LIN {X 0,Y 364.847,Z 1093.089,A -85,B 0,C 180,E1 16368.459,E2 16368.459} C_VEL
LIN {X 0,Y 364.189,Z 1097.02,A -85,B 0,C 180,E1 16366.666,E2 16366.666} C_VEL
LIN {X 0,Y 363.606,Z 1099.933,A -85,B 0,C 180,E1 16364.529,E2 16364.529} C_VEL
LIN {X 0,Y 363.242,Z 1100.889,A -85,B 0,C 180,E1 16362.54,E2 16362.54} C_VEL
LIN {X 0,Y 363.064,Z 1100.469,A -85,B 0,C 180,E1 16360.702,E2 16360.702} C_VEL
LIN {X 0,Y 363.041,Z 1098.768,A -85,B 0,C 180,E1 16358.85,E2 16358.85} C_VEL
LIN {X 0,Y 363.189,Z 1095.43,A -85,B 0,C 180,E1 16356.816,E2 16356.816} C_VEL
LIN {X 0,Y 363.562,Z 1089.731,A -85,B 0,C 180,E1 16354.593,E2 16354.593} C_VEL
LIN {X 0,Y 364.021,Z 1083.743,A -85,B 0,C 180,E1 16352.871,E2 16352.871} C_VEL
LIN {X 0,Y 364.565,Z 1076.974,A -85,B 0,C 180,E1 16351.316,E2 16351.316} C_VEL
LIN {X 0,Y 365.337,Z 1067.492,A -85,B 0,C 180,E1 16349.558,E2 16349.558} C_VEL
LIN {X 0,Y 366.143,Z 1056.281,A -85,B 0,C 180,E1 16347.95,E2 16347.95} C_VEL
LIN {X 0,Y 366.856,Z 1045.383,A -85,B 0,C 180,E1 16346.688,E2 16346.688} C_VEL
LIN {X 0,Y 366.982,Z 1044.003,A -85,B 0,C 180,E1 16346.513,E2 16346.513} C_VEL
LIN {X 0,Y 368.446,Z 1044.428,A -85,B 0,C 180,E1 16346.01,E2 16346.01} C_VEL
LIN {X 0,Y 371.071,Z 1043.748,A -85,B 0,C 180,E1 16345.537,E2 16345.537} C_VEL
LIN {X 0,Y 374.017,Z 1043.467,A -85,B 0,C 180,E1 16344.893,E2 16344.893} C_VEL
LIN {X 0,Y 377.167,Z 1042.77,A -85,B 0,C 180,E1 16344.322,E2 16344.322} C_VEL
LIN {X 0,Y 386.849,Z 1040.234,A -85,B 0,C 180,E1 16342.784,E2 16342.784} C_VEL
LIN {X 0,Y 400.514,Z 1035.789,A -85,B 0,C 180,E1 16341.014,E2 16341.014} C_VEL
LIN {X 0,Y 412.392,Z 1030.85,A -85,B 0,C 180,E1 16339.838,E2 16339.838} C_VEL
LIN {X 0,Y 415.714,Z 1029.331,A -85,B 0,C 180,E1 16339.543,E2 16339.543} C_VEL
LIN {X 0,Y 407.381,Z 1049.235,A -85,B 0,C 180,E1 16337.007,E2 16337.007} C_VEL
LIN {X 0,Y 399.448,Z 1067.755,A -85,B 0,C 180,E1 16334.282,E2 16334.282} C_VEL
LIN {X 0,Y 391.606,Z 1085.492,A -85,B 0,C 180,E1 16331.206,E2 16331.206} C_VEL
LIN {X 0,Y 384.418,Z 1102.08,A -85,B 0,C 180,E1 16327.87,E2 16327.87} C_VEL
LIN {X 0,Y 378.236,Z 1116.473,A -85,B 0,C 180,E1 16324.454,E2 16324.454} C_VEL
LIN {X 0,Y 372.918,Z 1129.743,A -85,B 0,C 180,E1 16320.807,E2 16320.807} C_VEL
LIN {X 0,Y 368.629,Z 1141.026,A -85,B 0,C 180,E1 16317.111,E2 16317.111} C_VEL
LIN {X 0,Y 365.504,Z 1150.37,A -85,B 0,C 180,E1 16313.543,E2 16313.543} C_VEL
LIN {X 0,Y 362.854,Z 1159.499,A -85,B 0,C 180,E1 16309.311,E2 16309.311} C_VEL
LIN {X 0,Y 361.475,Z 1165.476,A -85,B 0,C 180,E1 16305.895,E2 16305.895} C_VEL
LIN {X 0,Y 360.647,Z 1170.154,A -85,B 0,C 180,E1 16302.599,E2 16302.599} C_VEL
LIN {X 0,Y 360.167,Z 1174.441,A -85,B 0,C 180,E1 16298.624,E2 16298.624} C_VEL
LIN {X 0,Y 359.992,Z 1176.868,A -85,B 0,C 180,E1 16294.941,E2 16294.941} C_VEL
LIN {X 0,Y 359.958,Z 1177.939,A -85,B 0,C 180,E1 16291.753,E2 16291.753} C_VEL
LIN {X 0,Y 359.957,Z 1178.023,A -85,B 0,C 180,E1 16288.729,E2 16288.729} C_VEL
LIN {X 0,Y 359.981,Z 1177.183,A -85,B 0,C 180,E1 16285.689,E2 16285.689} C_VEL
LIN {X 0,Y 360.071,Z 1175.437,A -85,B 0,C 180,E1 16282.663,E2 16282.663} C_VEL
LIN {X 0,Y 360.313,Z 1172.766,A -85,B 0,C 180,E1 16279.61,E2 16279.61} C_VEL
LIN {X 0,Y 360.88,Z 1168.742,A -85,B 0,C 180,E1 16276.217,E2 16276.217} C_VEL
LIN {X 0,Y 361.623,Z 1164.805,A -85,B 0,C 180,E1 16273.586,E2 16273.586} C_VEL
LIN {X 0,Y 361.083,Z 1162.995,A -85,B 0,C 180,E1 16272.394,E2 16272.394} C_VEL
LIN {X 0,Y 356.335,Z 1157.659,A -85,B 0,C 180,E1 16269.097,E2 16269.097} C_VEL
LIN {X 0,Y 356.258,Z 1155.765,A -85,B 0,C 180,E1 16268.158,E2 16268.158} C_VEL
LIN {X 0,Y 358.806,Z 1148.037,A -85,B 0,C 180,E1 16264.765,E2 16264.765} C_VEL
LIN {X 0,Y 362.973,Z 1136.898,A -85,B 0,C 180,E1 16260.64,E2 16260.64} C_VEL
LIN {X 0,Y 367.709,Z 1125.312,A -85,B 0,C 180,E1 16257.057,E2 16257.057} C_VEL
LIN {X 0,Y 373.773,Z 1111.505,A -85,B 0,C 180,E1 16253.374,E2 16253.374} C_VEL
LIN {X 0,Y 380.314,Z 1096.941,A -85,B 0,C 180,E1 16250.099,E2 16250.099} C_VEL
LIN {X 0,Y 387.848,Z 1080.633,A -85,B 0,C 180,E1 16246.911,E2 16246.911} C_VEL
LIN {X 0,Y 395.874,Z 1062.8,A -85,B 0,C 180,E1 16243.962,E2 16243.962} C_VEL
LIN {X 0,Y 403.958,Z 1044.778,A -85,B 0,C 180,E1 16241.368,E2 16241.368} C_VEL
LIN {X 0,Y 412.483,Z 1024.657,A -85,B 0,C 180,E1 16238.914,E2 16238.914} C_VEL
LIN {X 0,Y 421.011,Z 1003.86,A -85,B 0,C 180,E1 16236.726,E2 16236.726} C_VEL
LIN {X 0,Y 429.064,Z 982.412,A -85,B 0,C 180,E1 16234.817,E2 16234.817} C_VEL
LIN {X 0,Y 436.879,Z 960.16,A -85,B 0,C 180,E1 16233.11,E2 16233.11} C_VEL
LIN {X 0,Y 443.975,Z 937.444,A -85,B 0,C 180,E1 16231.651,E2 16231.651} C_VEL
LIN {X 0,Y 450.439,Z 914.796,A -85,B 0,C 180,E1 16230.406,E2 16230.406} C_VEL
LIN {X 0,Y 456.319,Z 890.425,A -85,B 0,C 180,E1 16229.301,E2 16229.301} C_VEL
LIN {X 0,Y 461.547,Z 865.497,A -85,B 0,C 180,E1 16228.371,E2 16228.371} C_VEL
LIN {X 0,Y 467.573,Z 829.912,A -85,B 0,C 180,E1 16227.349,E2 16227.349} C_VEL
LIN {X 0,Y 480.681,Z 750.241,A -85,B 0,C 180,E1 16225.486,E2 16225.486} C_VEL
LIN {X 0,Y 491.44,Z 677.516,A -85,B 0,C 180,E1 16223.979,E2 16223.979} C_VEL
LIN {X 0,Y 500.182,Z 608.907,A -85,B 0,C 180,E1 16222.702,E2 16222.702} C_VEL
LIN {X 0,Y 506.001,Z 552.806,A -85,B 0,C 180,E1 16221.724,E2 16221.724} C_VEL
LIN {X 0,Y 502.096,Z 549.766,A -85,B 0,C 180,E1 16220.396,E2 16220.396} C_VEL
LIN {X 0,Y 494.551,Z 544.225,A -85,B 0,C 180,E1 16217.533,E2 16217.533} C_VEL
LIN {X 0,Y 486.719,Z 540.701,A -85,B 0,C 180,E1 16214.029,E2 16214.029} C_VEL
LIN {X 0,Y 480.667,Z 539.029,A -85,B 0,C 180,E1 16210.548,E2 16210.548} C_VEL
LIN {X 0,Y 479.161,Z 538.841,A -85,B 0,C 180,E1 16209.489,E2 16209.489} C_VEL
LIN {X 0,Y 474.514,Z 541.062,A -85,B 0,C 180,E1 16205.32,E2 16205.32} C_VEL
LIN {X 0,Y 472.587,Z 544.325,A -85,B 0,C 180,E1 16202.425,E2 16202.425} C_VEL
LIN {X 0,Y 471.775,Z 549.574,A -85,B 0,C 180,E1 16199.15,E2 16199.15} C_VEL
LIN {X 0,Y 474.61,Z 557.775,A -85,B 0,C 180,E1 16195.892,E2 16195.892} C_VEL
LIN {X 0,Y 476.871,Z 565.149,A -85,B 0,C 180,E1 16193.499,E2 16193.499} C_VEL
LIN {X 0,Y 472.618,Z 578.224,A -85,B 0,C 180,E1 16192.256,E2 16192.256} C_VEL
LIN {X 0,Y 471.814,Z 611.299,A -85,B 0,C 180,E1 16189.784,E2 16189.784} C_VEL
LIN {X 0,Y 471.576,Z 643.072,A -85,B 0,C 180,E1 16187.572,E2 16187.572} C_VEL
LIN {X 0,Y 471.999,Z 675.982,A -85,B 0,C 180,E1 16185.281,E2 16185.281} C_VEL
LIN {X 0,Y 473.232,Z 701.845,A -85,B 0,C 180,E1 16183.221,E2 16183.221} C_VEL
LIN {X 0,Y 475.279,Z 724.423,A -85,B 0,C 180,E1 16181.175,E2 16181.175} C_VEL
LIN {X 0,Y 477.851,Z 742.846,A -85,B 0,C 180,E1 16179.323,E2 16179.323} C_VEL
LIN {X 0,Y 481.269,Z 760.271,A -85,B 0,C 180,E1 16177.412,E2 16177.412} C_VEL
LIN {X 0,Y 486.893,Z 780.718,A -85,B 0,C 180,E1 16174.94,E2 16174.94} C_VEL
LIN {X 0,Y 486.96,Z 781.774,A -85,B 0,C 180,E1 16174.871,E2 16174.871} C_VEL
LIN {X 0,Y 480.312,Z 821.81,A -85,B 0,C 180,E1 16174.02,E2 16174.02} C_VEL
LIN {X 0,Y 472.503,Z 860.702,A -85,B 0,C 180,E1 16173.049,E2 16173.049} C_VEL
LIN {X 0,Y 464.769,Z 894.968,A -85,B 0,C 180,E1 16171.953,E2 16171.953} C_VEL
LIN {X 0,Y 456.674,Z 928.359,A -85,B 0,C 180,E1 16170.62,E2 16170.62} C_VEL
LIN {X 0,Y 448.577,Z 959.455,A -85,B 0,C 180,E1 16169.108,E2 16169.108} C_VEL
LIN {X 0,Y 440.535,Z 988.437,A -85,B 0,C 180,E1 16167.433,E2 16167.433} C_VEL
LIN {X 0,Y 433.872,Z 1010.028,A -85,B 0,C 180,E1 16165.943,E2 16165.943} C_VEL
LIN {X 0,Y 426.483,Z 1031.191,A -85,B 0,C 180,E1 16164.209,E2 16164.209} C_VEL
LIN {X 0,Y 419.044,Z 1050.358,A -85,B 0,C 180,E1 16162.349,E2 16162.349} C_VEL
LIN {X 0,Y 411.17,Z 1069.3,A -85,B 0,C 180,E1 16160.211,E2 16160.211} C_VEL
LIN {X 0,Y 402.736,Z 1088.062,A -85,B 0,C 180,E1 16157.716,E2 16157.716} C_VEL
LIN {X 0,Y 394.452,Z 1105.313,A -85,B 0,C 180,E1 16154.989,E2 16154.989} C_VEL
LIN {X 0,Y 386.613,Z 1120.941,A -85,B 0,C 180,E1 16152.075,E2 16152.075} C_VEL
LIN {X 0,Y 378.836,Z 1136.107,A -85,B 0,C 180,E1 16148.718,E2 16148.718} C_VEL
LIN {X 0,Y 371.928,Z 1149.46,A -85,B 0,C 180,E1 16145.187,E2 16145.187} C_VEL
LIN {X 0,Y 365.978,Z 1161.24,A -85,B 0,C 180,E1 16141.452,E2 16141.452} C_VEL
LIN {X 0,Y 360.912,Z 1171.835,A -85,B 0,C 180,E1 16137.378,E2 16137.378} C_VEL
LIN {X 0,Y 357.016,Z 1180.868,A -85,B 0,C 180,E1 16133.082,E2 16133.082} C_VEL
LIN {X 0,Y 354.391,Z 1188.078,A -85,B 0,C 180,E1 16128.76,E2 16128.76} C_VEL
LIN {X 0,Y 352.869,Z 1193.636,A -85,B 0,C 180,E1 16124.437,E2 16124.437} C_VEL
LIN {X 0,Y 352.161,Z 1197.659,A -85,B 0,C 180,E1 16120.137,E2 16120.137} C_VEL
LIN {X 0,Y 351.969,Z 1200.163,A -85,B 0,C 180,E1 16116.031,E2 16116.031} C_VEL
LIN {X 0,Y 351.957,Z 1201.387,A -85,B 0,C 180,E1 16112.115,E2 16112.115} C_VEL
LIN {X 0,Y 351.961,Z 1201.43,A -85,B 0,C 180,E1 16108.37,E2 16108.37} C_VEL
LIN {X 0,Y 351.963,Z 1200.374,A -85,B 0,C 180,E1 16104.455,E2 16104.455} C_VEL
LIN {X 0,Y 352.107,Z 1198.172,A -85,B 0,C 180,E1 16100.518,E2 16100.518} C_VEL
LIN {X 0,Y 352.708,Z 1194.383,A -85,B 0,C 180,E1 16096.222,E2 16096.222} C_VEL
LIN {X 0,Y 354.091,Z 1189.033,A -85,B 0,C 180,E1 16091.902,E2 16091.902} C_VEL
LIN {X 0,Y 356.533,Z 1182.047,A -85,B 0,C 180,E1 16087.577,E2 16087.577} C_VEL
LIN {X 0,Y 360.222,Z 1173.286,A -85,B 0,C 180,E1 16083.276,E2 16083.276} C_VEL
LIN {X 0,Y 365.081,Z 1163.008,A -85,B 0,C 180,E1 16079.191,E2 16079.191} C_VEL
LIN {X 0,Y 371.267,Z 1150.699,A -85,B 0,C 180,E1 16075.181,E2 16075.181} C_VEL
LIN {X 0,Y 378.516,Z 1136.712,A -85,B 0,C 180,E1 16071.432,E2 16071.432} C_VEL
LIN {X 0,Y 386.202,Z 1121.734,A -85,B 0,C 180,E1 16068.088,E2 16068.088} C_VEL
LIN {X 0,Y 394.075,Z 1106.054,A -85,B 0,C 180,E1 16065.139,E2 16065.139} C_VEL
LIN {X 0,Y 402.703,Z 1088.053,A -85,B 0,C 180,E1 16062.29,E2 16062.29} C_VEL
LIN {X 0,Y 410.926,Z 1069.744,A -85,B 0,C 180,E1 16059.851,E2 16059.851} C_VEL
LIN {X 0,Y 419.14,Z 1050.106,A -85,B 0,C 180,E1 16057.625,E2 16057.625} C_VEL
LIN {X 0,Y 427.021,Z 1029.58,A -85,B 0,C 180,E1 16055.656,E2 16055.656} C_VEL
LIN {X 0,Y 434.714,Z 1007.363,A -85,B 0,C 180,E1 16053.865,E2 16053.865} C_VEL
LIN {X 0,Y 441.705,Z 984.375,A -85,B 0,C 180,E1 16052.316,E2 16052.316} C_VEL
LIN {X 0,Y 450.4,Z 952.387,A -85,B 0,C 180,E1 16050.529,E2 16050.529} C_VEL
LIN {X 0,Y 458.422,Z 921.073,A -85,B 0,C 180,E1 16049.07,E2 16049.07} C_VEL
LIN {X 0,Y 466.669,Z 886.521,A -85,B 0,C 180,E1 16047.759,E2 16047.759} C_VEL
LIN {X 0,Y 474.383,Z 851.48,A -85,B 0,C 180,E1 16046.708,E2 16046.708} C_VEL
LIN {X 0,Y 482.278,Z 810.288,A -85,B 0,C 180,E1 16045.722,E2 16045.722} C_VEL
LIN {X 0,Y 488.506,Z 769.42,A -85,B 0,C 180,E1 16044.887,E2 16044.887} C_VEL
LIN {X 0,Y 493.484,Z 727.631,A -85,B 0,C 180,E1 16044.188,E2 16044.188} C_VEL
LIN {X 0,Y 498.328,Z 671.925,A -85,B 0,C 180,E1 16043.44,E2 16043.44} C_VEL
LIN {X 0,Y 501.803,Z 632.657,A -85,B 0,C 180,E1 16042.905,E2 16042.905} C_VEL
LIN {X 0,Y 505.015,Z 611.369,A -85,B 0,C 180,E1 16042.605,E2 16042.605} C_VEL
LIN {X 0,Y 498.401,Z 626.921,A -85,B 0,C 180,E1 16041.748,E2 16041.748} C_VEL
LIN {X 0,Y 492.948,Z 644.379,A -85,B 0,C 180,E1 16040.916,E2 16040.916} C_VEL
LIN {X 0,Y 489.241,Z 656.284,A -85,B 0,C 180,E1 16040.254,E2 16040.254} C_VEL
LIN {X 0,Y 483.115,Z 679.417,A -85,B 0,C 180,E1 16039.229,E2 16039.229} C_VEL
LIN {X 0,Y 477.477,Z 698.025,A -85,B 0,C 180,E1 16038.181,E2 16038.181} C_VEL
LIN {X 0,Y 470.537,Z 721.804,A -85,B 0,C 180,E1 16037.085,E2 16037.085} C_VEL
LIN {X 0,Y 464.748,Z 738.439,A -85,B 0,C 180,E1 16036.081,E2 16036.081} C_VEL
LIN {X 0,Y 457.916,Z 758.928,A -85,B 0,C 180,E1 16035.069,E2 16035.069} C_VEL
LIN {X 0,Y 451.933,Z 774.644,A -85,B 0,C 180,E1 16034.069,E2 16034.069} C_VEL
LIN {X 0,Y 445.663,Z 791.698,A -85,B 0,C 180,E1 16033.14,E2 16033.14} C_VEL
LIN {X 0,Y 440.732,Z 803.817,A -85,B 0,C 180,E1 16032.305,E2 16032.305} C_VEL
LIN {X 0,Y 434.442,Z 819.965,A -85,B 0,C 180,E1 16031.356,E2 16031.356} C_VEL
LIN {X 0,Y 430.125,Z 830.145,A -85,B 0,C 180,E1 16030.605,E2 16030.605} C_VEL
LIN {X 0,Y 424.219,Z 844.754,A -85,B 0,C 180,E1 16029.693,E2 16029.693} C_VEL
LIN {X 0,Y 420.064,Z 854.369,A -85,B 0,C 180,E1 16028.941,E2 16028.941} C_VEL
LIN {X 0,Y 414.446,Z 867.955,A -85,B 0,C 180,E1 16028.044,E2 16028.044} C_VEL
LIN {X 0,Y 411.21,Z 875.316,A -85,B 0,C 180,E1 16027.405,E2 16027.405} C_VEL
LIN {X 0,Y 405.131,Z 890.099,A -85,B 0,C 180,E1 16026.519,E2 16026.519} C_VEL
LIN {X 0,Y 401.582,Z 898.618,A -85,B 0,C 180,E1 16025.891,E2 16025.891} C_VEL
LIN {X 0,Y 397.183,Z 909.858,A -85,B 0,C 180,E1 16025.417,E2 16025.417} C_VEL
LIN {X 0,Y 393.369,Z 919.051,A -85,B 0,C 180,E1 16024.846,E2 16024.846} C_VEL
LIN {X 0,Y 388.804,Z 930.174,A -85,B 0,C 180,E1 16024.351,E2 16024.351} C_VEL
LIN {X 0,Y 385.071,Z 938.389,A -85,B 0,C 180,E1 16023.767,E2 16023.767} C_VEL
LIN {X 0,Y 380.587,Z 947.982,A -85,B 0,C 180,E1 16023.277,E2 16023.277} C_VEL
LIN {X 0,Y 377.253,Z 954.474,A -85,B 0,C 180,E1 16022.735,E2 16022.735} C_VEL
LIN {X 0,Y 373.263,Z 962.133,A -85,B 0,C 180,E1 16022.29,E2 16022.29} C_VEL
LIN {X 0,Y 370.135,Z 967.7,A -85,B 0,C 180,E1 16021.734,E2 16021.734} C_VEL
LIN {X 0,Y 367.076,Z 973.213,A -85,B 0,C 180,E1 16021.402,E2 16021.402} C_VEL
LIN {X 0,Y 364.777,Z 976.956,A -85,B 0,C 180,E1 16020.942,E2 16020.942} C_VEL
LIN {X 0,Y 364.255,Z 978.134,A -85,B 0,C 180,E1 16020.767,E2 16020.767} C_VEL
LIN {X 0,Y 364.021,Z 1008.238,A -85,B 0,C 180,E1 16019.887,E2 16019.887} C_VEL
LIN {X 0,Y 363.779,Z 1022.911,A -85,B 0,C 180,E1 16019.213,E2 16019.213} C_VEL
LIN {X 0,Y 363.148,Z 1036.96,A -85,B 0,C 180,E1 16018.264,E2 16018.264} C_VEL
LIN {X 0,Y 362.477,Z 1047.823,A -85,B 0,C 180,E1 16017.312,E2 16017.312} C_VEL
LIN {X 0,Y 361.55,Z 1059.449,A -85,B 0,C 180,E1 16016.035,E2 16016.035} C_VEL
LIN {X 0,Y 360.369,Z 1070.638,A -85,B 0,C 180,E1 16014.427,E2 16014.427} C_VEL
LIN {X 0,Y 359.394,Z 1078.737,A -85,B 0,C 180,E1 16012.968,E2 16012.968} C_VEL
LIN {X 0,Y 358.414,Z 1085.979,A -85,B 0,C 180,E1 16011.336,E2 16011.336} C_VEL
LIN {X 0,Y 357.301,Z 1093.047,A -85,B 0,C 180,E1 16009.193,E2 16009.193} C_VEL
LIN {X 0,Y 356.534,Z 1097.282,A -85,B 0,C 180,E1 16007.364,E2 16007.364} C_VEL
LIN {X 0,Y 355.984,Z 1099.939,A -85,B 0,C 180,E1 16005.69,E2 16005.69} C_VEL
LIN {X 0,Y 355.568,Z 1101.514,A -85,B 0,C 180,E1 16004.003,E2 16004.003} C_VEL
LIN {X 0,Y 355.29,Z 1102.035,A -85,B 0,C 180,E1 16002.305,E2 16002.305} C_VEL
LIN {X 0,Y 355.133,Z 1101.492,A -85,B 0,C 180,E1 16000.595,E2 16000.595} C_VEL
LIN {X 0,Y 355.114,Z 1099.658,A -85,B 0,C 180,E1 15998.702,E2 15998.702} C_VEL
LIN {X 0,Y 355.302,Z 1095.778,A -85,B 0,C 180,E1 15996.446,E2 15996.446} C_VEL
LIN {X 0,Y 355.641,Z 1090.642,A -85,B 0,C 180,E1 15994.491,E2 15994.491} C_VEL
LIN {X 0,Y 356.105,Z 1084.712,A -85,B 0,C 180,E1 15992.762,E2 15992.762} C_VEL
LIN {X 0,Y 356.745,Z 1077.037,A -85,B 0,C 180,E1 15990.986,E2 15990.986} C_VEL
LIN {X 0,Y 357.62,Z 1066.194,A -85,B 0,C 180,E1 15989.039,E2 15989.039} C_VEL
LIN {X 0,Y 358.301,Z 1057.113,A -85,B 0,C 180,E1 15987.735,E2 15987.735} C_VEL
LIN {X 0,Y 358.794,Z 1050.317,A -85,B 0,C 180,E1 15986.892,E2 15986.892} C_VEL
LIN {X 0,Y 359.947,Z 1050.8,A -85,B 0,C 180,E1 15986.441,E2 15986.441} C_VEL
LIN {X 0,Y 362.931,Z 1050.277,A -85,B 0,C 180,E1 15985.804,E2 15985.804} C_VEL
LIN {X 0,Y 366.425,Z 1049.857,A -85,B 0,C 180,E1 15985.037,E2 15985.037} C_VEL
LIN {X 0,Y 371.457,Z 1048.964,A -85,B 0,C 180,E1 15984.069,E2 15984.069} C_VEL
LIN {X 0,Y 381.641,Z 1046.625,A -85,B 0,C 180,E1 15982.377,E2 15982.377} C_VEL
LIN {X 0,Y 397.716,Z 1041.548,A -85,B 0,C 180,E1 15980.314,E2 15980.314} C_VEL
LIN {X 0,Y 406.743,Z 1038.116,A -85,B 0,C 180,E1 15979.377,E2 15979.377} C_VEL
LIN {X 0,Y 398.216,Z 1057.629,A -85,B 0,C 180,E1 15976.735,E2 15976.735} C_VEL
LIN {X 0,Y 390.284,Z 1075.058,A -85,B 0,C 180,E1 15973.953,E2 15973.953} C_VEL
LIN {X 0,Y 382.54,Z 1092.131,A -85,B 0,C 180,E1 15970.804,E2 15970.804} C_VEL
LIN {X 0,Y 375.579,Z 1107.339,A -85,B 0,C 180,E1 15967.499,E2 15967.499} C_VEL
LIN {X 0,Y 369.302,Z 1121.638,A -85,B 0,C 180,E1 15963.902,E2 15963.902} C_VEL
LIN {X 0,Y 364.055,Z 1134.074,A -85,B 0,C 180,E1 15960.175,E2 15960.175} C_VEL
LIN {X 0,Y 359.932,Z 1144.921,A -85,B 0,C 180,E1 15956.392,E2 15956.392} C_VEL
LIN {X 0,Y 356.699,Z 1154.354,A -85,B 0,C 180,E1 15952.412,E2 15952.412} C_VEL
LIN {X 0,Y 354.688,Z 1161.281,A -85,B 0,C 180,E1 15948.918,E2 15948.918} C_VEL
LIN {X 0,Y 353.214,Z 1167.787,A -85,B 0,C 180,E1 15944.93,E2 15944.93} C_VEL
LIN {X 0,Y 352.386,Z 1172.767,A -85,B 0,C 180,E1 15940.796,E2 15940.796} C_VEL
LIN {X 0,Y 352.098,Z 1175.63,A -85,B 0,C 180,E1 15937.508,E2 15937.508} C_VEL
LIN {X 0,Y 351.986,Z 1177.423,A -85,B 0,C 180,E1 15934.368,E2 15934.368} C_VEL
LIN {X 0,Y 351.963,Z 1178.271,A -85,B 0,C 180,E1 15931.304,E2 15931.304} C_VEL
LIN {X 0,Y 351.963,Z 1178.216,A -85,B 0,C 180,E1 15928.211,E2 15928.211} C_VEL
LIN {X 0,Y 352,Z 1177.172,A -85,B 0,C 180,E1 15924.95,E2 15924.95} C_VEL
LIN {X 0,Y 352.198,Z 1174.647,A -85,B 0,C 180,E1 15921.019,E2 15921.019} C_VEL
LIN {X 0,Y 352.714,Z 1170.464,A -85,B 0,C 180,E1 15917.061,E2 15917.061} C_VEL
LIN {X 0,Y 353.584,Z 1165.887,A -85,B 0,C 180,E1 15913.745,E2 15913.745} C_VEL
LIN {X 0,Y 355.059,Z 1159.936,A -85,B 0,C 180,E1 15910.251,E2 15910.251} C_VEL
LIN {X 0,Y 356.258,Z 1155.765,A -85,B 0,C 180,E1 15908.158,E2 15908.158} C_VEL
LIN {X 0,Y 356.062,Z 1153.422,A -85,B 0,C 180,E1 15906.968,E2 15906.968} C_VEL
LIN {X 0,Y 352.486,Z 1147.135,A -85,B 0,C 180,E1 15903.731,E2 15903.731} C_VEL
LIN {X 0,Y 352.706,Z 1144.684,A -85,B 0,C 180,E1 15902.723,E2 15902.723} C_VEL
LIN {X 0,Y 356.777,Z 1134.636,A -85,B 0,C 180,E1 15899.148,E2 15899.148} C_VEL
LIN {X 0,Y 362.322,Z 1122.162,A -85,B 0,C 180,E1 15895.324,E2 15895.324} C_VEL
LIN {X 0,Y 368.965,Z 1107.76,A -85,B 0,C 180,E1 15891.644,E2 15891.644} C_VEL
LIN {X 0,Y 376.468,Z 1092.113,A -85,B 0,C 180,E1 15888.194,E2 15888.194} C_VEL
LIN {X 0,Y 384.204,Z 1075.734,A -85,B 0,C 180,E1 15885.152,E2 15885.152} C_VEL
LIN {X 0,Y 392.628,Z 1058.004,A -85,B 0,C 180,E1 15882.289,E2 15882.289} C_VEL
LIN {X 0,Y 401.097,Z 1039.274,A -85,B 0,C 180,E1 15879.735,E2 15879.735} C_VEL
LIN {X 0,Y 409.723,Z 1019.733,A -85,B 0,C 180,E1 15877.421,E2 15877.421} C_VEL
LIN {X 0,Y 418.234,Z 998.835,A -85,B 0,C 180,E1 15875.325,E2 15875.325} C_VEL
LIN {X 0,Y 426.607,Z 977.15,A -85,B 0,C 180,E1 15873.451,E2 15873.451} C_VEL
LIN {X 0,Y 434.28,Z 954.935,A -85,B 0,C 180,E1 15871.838,E2 15871.838} C_VEL
LIN {X 0,Y 441.644,Z 931.739,A -85,B 0,C 180,E1 15870.396,E2 15870.396} C_VEL
LIN {X 0,Y 447.919,Z 908.835,A -85,B 0,C 180,E1 15869.216,E2 15869.216} C_VEL
LIN {X 0,Y 453.727,Z 885.041,A -85,B 0,C 180,E1 15868.182,E2 15868.182} C_VEL
LIN {X 0,Y 458.651,Z 860.14,A -85,B 0,C 180,E1 15867.318,E2 15867.318} C_VEL
LIN {X 0,Y 465.852,Z 818.765,A -85,B 0,C 180,E1 15866.189,E2 15866.189} C_VEL
LIN {X 0,Y 478.662,Z 742.339,A -85,B 0,C 180,E1 15864.436,E2 15864.436} C_VEL
LIN {X 0,Y 489.296,Z 671.078,A -85,B 0,C 180,E1 15862.983,E2 15862.983} C_VEL
LIN {X 0,Y 497.897,Z 603.539,A -85,B 0,C 180,E1 15861.747,E2 15861.747} C_VEL
LIN {X 0,Y 502.624,Z 558.958,A -85,B 0,C 180,E1 15860.983,E2 15860.983} C_VEL
LIN {X 0,Y 493.285,Z 552.098,A -85,B 0,C 180,E1 15857.457,E2 15857.457} C_VEL
LIN {X 0,Y 485.529,Z 548.598,A -85,B 0,C 180,E1 15853.943,E2 15853.943} C_VEL
LIN {X 0,Y 479.529,Z 546.942,A -85,B 0,C 180,E1 15850.452,E2 15850.452} C_VEL
LIN {X 0,Y 478.022,Z 546.893,A -85,B 0,C 180,E1 15849.39,E2 15849.39} C_VEL
LIN {X 0,Y 473.639,Z 548.943,A -85,B 0,C 180,E1 15845.451,E2 15845.451} C_VEL
LIN {X 0,Y 471.657,Z 552.219,A -85,B 0,C 180,E1 15842.552,E2 15842.552} C_VEL
LIN {X 0,Y 470.67,Z 557.64,A -85,B 0,C 180,E1 15839.209,E2 15839.209} C_VEL
LIN {X 0,Y 471.157,Z 566.416,A -85,B 0,C 180,E1 15835.435,E2 15835.435} C_VEL
LIN {X 0,Y 471.815,Z 570.474,A -85,B 0,C 180,E1 15834.009,E2 15834.009} C_VEL
LIN {X 0,Y 470.347,Z 606.661,A -85,B 0,C 180,E1 15831.238,E2 15831.238} C_VEL
LIN {X 0,Y 469.737,Z 637.417,A -85,B 0,C 180,E1 15829.041,E2 15829.041} C_VEL
LIN {X 0,Y 469.675,Z 678.234,A -85,B 0,C 180,E1 15826.206,E2 15826.206} C_VEL
LIN {X 0,Y 470.456,Z 703.471,A -85,B 0,C 180,E1 15824.198,E2 15824.198} C_VEL
LIN {X 0,Y 472.198,Z 727.784,A -85,B 0,C 180,E1 15822.007,E2 15822.007} C_VEL
LIN {X 0,Y 474.682,Z 747.616,A -85,B 0,C 180,E1 15819.999,E2 15819.999} C_VEL
LIN {X 0,Y 477.933,Z 765.694,A -85,B 0,C 180,E1 15817.991,E2 15817.991} C_VEL
LIN {X 0,Y 482.757,Z 785.128,A -85,B 0,C 180,E1 15815.655,E2 15815.655} C_VEL
LIN {X 0,Y 475.629,Z 826.544,A -85,B 0,C 180,E1 15814.758,E2 15814.758} C_VEL
LIN {X 0,Y 467.217,Z 866.338,A -85,B 0,C 180,E1 15813.733,E2 15813.733} C_VEL
LIN {X 0,Y 459.218,Z 900.735,A -85,B 0,C 180,E1 15812.596,E2 15812.596} C_VEL
LIN {X 0,Y 450.937,Z 933.757,A -85,B 0,C 180,E1 15811.238,E2 15811.238} C_VEL
LIN {X 0,Y 442.195,Z 966.242,A -85,B 0,C 180,E1 15809.61,E2 15809.61} C_VEL
LIN {X 0,Y 434.459,Z 992.997,A -85,B 0,C 180,E1 15808.012,E2 15808.012} C_VEL
LIN {X 0,Y 427.188,Z 1014.841,A -85,B 0,C 180,E1 15806.431,E2 15806.431} C_VEL
LIN {X 0,Y 419.377,Z 1035.953,A -85,B 0,C 180,E1 15804.623,E2 15804.623} C_VEL
LIN {X 0,Y 411.379,Z 1055.622,A -85,B 0,C 180,E1 15802.632,E2 15802.632} C_VEL
LIN {X 0,Y 402.8,Z 1075.114,A -85,B 0,C 180,E1 15800.308,E2 15800.308} C_VEL
LIN {X 0,Y 394.043,Z 1093.467,A -85,B 0,C 180,E1 15797.701,E2 15797.701} C_VEL
LIN {X 0,Y 385.868,Z 1109.695,A -85,B 0,C 180,E1 15794.974,E2 15794.974} C_VEL
LIN {X 0,Y 377.946,Z 1124.931,A -85,B 0,C 180,E1 15791.977,E2 15791.977} C_VEL
LIN {X 0,Y 370.252,Z 1139.377,A -85,B 0,C 180,E1 15788.593,E2 15788.593} C_VEL
LIN {X 0,Y 362.945,Z 1152.926,A -85,B 0,C 180,E1 15784.766,E2 15784.766} C_VEL
LIN {X 0,Y 356.957,Z 1164.386,A -85,B 0,C 180,E1 15780.835,E2 15780.835} C_VEL
LIN {X 0,Y 352.067,Z 1174.382,A -85,B 0,C 180,E1 15776.659,E2 15776.659} C_VEL
LIN {X 0,Y 348.378,Z 1182.882,A -85,B 0,C 180,E1 15772.26,E2 15772.26} C_VEL
LIN {X 0,Y 345.885,Z 1189.844,A -85,B 0,C 180,E1 15767.668,E2 15767.668} C_VEL
LIN {X 0,Y 344.588,Z 1194.898,A -85,B 0,C 180,E1 15763.25,E2 15763.25} C_VEL
LIN {X 0,Y 344.078,Z 1198.343,A -85,B 0,C 180,E1 15759.026,E2 15759.026} C_VEL
LIN {X 0,Y 343.959,Z 1200.392,A -85,B 0,C 180,E1 15755.001,E2 15755.001} C_VEL
LIN {X 0,Y 343.968,Z 1201.21,A -85,B 0,C 180,E1 15751.164,E2 15751.164} C_VEL
LIN {X 0,Y 343.96,Z 1200.988,A -85,B 0,C 180,E1 15747.165,E2 15747.165} C_VEL
LIN {X 0,Y 343.981,Z 1199.676,A -85,B 0,C 180,E1 15743.321,E2 15743.321} C_VEL
LIN {X 0,Y 344.216,Z 1197.112,A -85,B 0,C 180,E1 15739.284,E2 15739.284} C_VEL
LIN {X 0,Y 345.066,Z 1192.836,A -85,B 0,C 180,E1 15734.781,E2 15734.781} C_VEL
LIN {X 0,Y 346.836,Z 1186.971,A -85,B 0,C 180,E1 15730.286,E2 15730.286} C_VEL
LIN {X 0,Y 349.767,Z 1179.507,A -85,B 0,C 180,E1 15725.869,E2 15725.869} C_VEL
LIN {X 0,Y 353.862,Z 1170.614,A -85,B 0,C 180,E1 15721.658,E2 15721.658} C_VEL
LIN {X 0,Y 359.362,Z 1159.711,A -85,B 0,C 180,E1 15717.466,E2 15717.466} C_VEL
LIN {X 0,Y 366.141,Z 1146.948,A -85,B 0,C 180,E1 15713.462,E2 15713.462} C_VEL
LIN {X 0,Y 373.287,Z 1133.598,A -85,B 0,C 180,E1 15709.992,E2 15709.992} C_VEL
LIN {X 0,Y 381.506,Z 1118.142,A -85,B 0,C 180,E1 15706.631,E2 15706.631} C_VEL
LIN {X 0,Y 390.07,Z 1101.477,A -85,B 0,C 180,E1 15703.594,E2 15703.594} C_VEL
LIN {X 0,Y 398.668,Z 1083.852,A -85,B 0,C 180,E1 15700.89,E2 15700.89} C_VEL
LIN {X 0,Y 407.291,Z 1065.053,A -85,B 0,C 180,E1 15698.45,E2 15698.45} C_VEL
LIN {X 0,Y 415.845,Z 1044.765,A -85,B 0,C 180,E1 15696.235,E2 15696.235} C_VEL
LIN {X 0,Y 424.095,Z 1023.384,A -85,B 0,C 180,E1 15694.27,E2 15694.27} C_VEL
LIN {X 0,Y 431.812,Z 1001.111,A -85,B 0,C 180,E1 15692.554,E2 15692.554} C_VEL
LIN {X 0,Y 438.891,Z 977.857,A -85,B 0,C 180,E1 15691.06,E2 15691.06} C_VEL
LIN {X 0,Y 447.269,Z 947.202,A -85,B 0,C 180,E1 15689.41,E2 15689.41} C_VEL
LIN {X 0,Y 455.488,Z 915.583,A -85,B 0,C 180,E1 15687.987,E2 15687.987} C_VEL
LIN {X 0,Y 463.724,Z 881.34,A -85,B 0,C 180,E1 15686.736,E2 15686.736} C_VEL
LIN {X 0,Y 471.448,Z 846.648,A -85,B 0,C 180,E1 15685.737,E2 15685.737} C_VEL
LIN {X 0,Y 479.592,Z 804.108,A -85,B 0,C 180,E1 15684.74,E2 15684.74} C_VEL
LIN {X 0,Y 486.2,Z 760.447,A -85,B 0,C 180,E1 15683.88,E2 15683.88} C_VEL
LIN {X 0,Y 490.991,Z 719.594,A -85,B 0,C 180,E1 15683.229,E2 15683.229} C_VEL
LIN {X 0,Y 495.062,Z 673.134,A -85,B 0,C 180,E1 15682.604,E2 15682.604} C_VEL
LIN {X 0,Y 497.855,Z 639.22,A -85,B 0,C 180,E1 15682.142,E2 15682.142} C_VEL
LIN {X 0,Y 491.97,Z 657.749,A -85,B 0,C 180,E1 15681.147,E2 15681.147} C_VEL
LIN {X 0,Y 485.087,Z 683.165,A -85,B 0,C 180,E1 15680.033,E2 15680.033} C_VEL
LIN {X 0,Y 479.245,Z 701.986,A -85,B 0,C 180,E1 15678.987,E2 15678.987} C_VEL
LIN {X 0,Y 472.552,Z 724.551,A -85,B 0,C 180,E1 15677.971,E2 15677.971} C_VEL
LIN {X 0,Y 466.473,Z 741.716,A -85,B 0,C 180,E1 15676.965,E2 15676.965} C_VEL
LIN {X 0,Y 459.006,Z 763.466,A -85,B 0,C 180,E1 15675.89,E2 15675.89} C_VEL
LIN {X 0,Y 453.101,Z 778.565,A -85,B 0,C 180,E1 15674.947,E2 15674.947} C_VEL
LIN {X 0,Y 446.565,Z 795.872,A -85,B 0,C 180,E1 15674.011,E2 15674.011} C_VEL
LIN {X 0,Y 441.654,Z 807.624,A -85,B 0,C 180,E1 15673.215,E2 15673.215} C_VEL
LIN {X 0,Y 435.08,Z 823.938,A -85,B 0,C 180,E1 15672.267,E2 15672.267} C_VEL
LIN {X 0,Y 430.709,Z 834.059,A -85,B 0,C 180,E1 15671.537,E2 15671.537} C_VEL
LIN {X 0,Y 424.464,Z 849.052,A -85,B 0,C 180,E1 15670.605,E2 15670.605} C_VEL
LIN {X 0,Y 420.302,Z 858.366,A -85,B 0,C 180,E1 15669.894,E2 15669.894} C_VEL
LIN {X 0,Y 414.601,Z 871.731,A -85,B 0,C 180,E1 15669.019,E2 15669.019} C_VEL
LIN {X 0,Y 411.218,Z 879.267,A -85,B 0,C 180,E1 15668.389,E2 15668.389} C_VEL
LIN {X 0,Y 404.604,Z 894.852,A -85,B 0,C 180,E1 15667.448,E2 15667.448} C_VEL
LIN {X 0,Y 401.672,Z 901.668,A -85,B 0,C 180,E1 15666.96,E2 15666.96} C_VEL
LIN {X 0,Y 396.435,Z 914.404,A -85,B 0,C 180,E1 15666.402,E2 15666.402} C_VEL
LIN {X 0,Y 393.358,Z 921.673,A -85,B 0,C 180,E1 15665.954,E2 15665.954} C_VEL
LIN {X 0,Y 388.629,Z 932.844,A -85,B 0,C 180,E1 15665.463,E2 15665.463} C_VEL
LIN {X 0,Y 384.344,Z 942.054,A -85,B 0,C 180,E1 15664.857,E2 15664.857} C_VEL
LIN {X 0,Y 379.905,Z 951.175,A -85,B 0,C 180,E1 15664.377,E2 15664.377} C_VEL
LIN {X 0,Y 376.834,Z 956.935,A -85,B 0,C 180,E1 15663.893,E2 15663.893} C_VEL
LIN {X 0,Y 372.641,Z 964.78,A -85,B 0,C 180,E1 15663.451,E2 15663.451} C_VEL
LIN {X 0,Y 368.927,Z 971.218,A -85,B 0,C 180,E1 15662.867,E2 15662.867} C_VEL
LIN {X 0,Y 365.299,Z 977.393,A -85,B 0,C 180,E1 15662.445,E2 15662.445} C_VEL
LIN {X 0,Y 362.621,Z 981.657,A -85,B 0,C 180,E1 15661.926,E2 15661.926} C_VEL
LIN {X 0,Y 359.563,Z 986.665,A -85,B 0,C 180,E1 15661.594,E2 15661.594} C_VEL
LIN {X 0,Y 357.274,Z 990.044,A -85,B 0,C 180,E1 15661.123,E2 15661.123} C_VEL
LIN {X 0,Y 356.859,Z 990.897,A -85,B 0,C 180,E1 15660.978,E2 15660.978} C_VEL
LIN {X 0,Y 356.73,Z 1011.349,A -85,B 0,C 180,E1 15660.311,E2 15660.311} C_VEL
LIN {X 0,Y 356.348,Z 1026.961,A -85,B 0,C 180,E1 15659.518,E2 15659.518} C_VEL
LIN {X 0,Y 355.723,Z 1039.389,A -85,B 0,C 180,E1 15658.631,E2 15658.631} C_VEL
LIN {X 0,Y 354.952,Z 1050.887,A -85,B 0,C 180,E1 15657.578,E2 15657.578} C_VEL
LIN {X 0,Y 353.795,Z 1063.463,A -85,B 0,C 180,E1 15656.082,E2 15656.082} C_VEL
LIN {X 0,Y 352.826,Z 1071.984,A -85,B 0,C 180,E1 15654.797,E2 15654.797} C_VEL
LIN {X 0,Y 351.778,Z 1080.008,A -85,B 0,C 180,E1 15653.308,E2 15653.308} C_VEL
LIN {X 0,Y 350.717,Z 1087.314,A -85,B 0,C 180,E1 15651.615,E2 15651.615} C_VEL
LIN {X 0,Y 349.547,Z 1094.279,A -85,B 0,C 180,E1 15649.451,E2 15649.451} C_VEL
LIN {X 0,Y 348.728,Z 1098.507,A -85,B 0,C 180,E1 15647.582,E2 15647.582} C_VEL
LIN {X 0,Y 348.14,Z 1101.15,A -85,B 0,C 180,E1 15645.87,E2 15645.87} C_VEL
LIN {X 0,Y 347.69,Z 1102.699,A -85,B 0,C 180,E1 15644.145,E2 15644.145} C_VEL
LIN {X 0,Y 347.373,Z 1103.185,A -85,B 0,C 180,E1 15642.322,E2 15642.322} C_VEL
LIN {X 0,Y 347.202,Z 1102.507,A -85,B 0,C 180,E1 15640.484,E2 15640.484} C_VEL
LIN {X 0,Y 347.198,Z 1100.328,A -85,B 0,C 180,E1 15638.369,E2 15638.369} C_VEL
LIN {X 0,Y 347.411,Z 1095.977,A -85,B 0,C 180,E1 15636.058,E2 15636.058} C_VEL
LIN {X 0,Y 347.773,Z 1090.828,A -85,B 0,C 180,E1 15634.15,E2 15634.15} C_VEL
LIN {X 0,Y 348.309,Z 1084.285,A -85,B 0,C 180,E1 15632.286,E2 15632.286} C_VEL
LIN {X 0,Y 349.109,Z 1074.794,A -85,B 0,C 180,E1 15630.21,E2 15630.21} C_VEL
LIN {X 0,Y 349.888,Z 1065.203,A -85,B 0,C 180,E1 15628.564,E2 15628.564} C_VEL
LIN {X 0,Y 350.592,Z 1056.457,A -85,B 0,C 180,E1 15627.3,E2 15627.3} C_VEL
LIN {X 0,Y 351.99,Z 1056.91,A -85,B 0,C 180,E1 15626.753,E2 15626.753} C_VEL
LIN {X 0,Y 354.827,Z 1056.546,A -85,B 0,C 180,E1 15626.085,E2 15626.085} C_VEL
LIN {X 0,Y 362.481,Z 1055.57,A -85,B 0,C 180,E1 15624.406,E2 15624.406} C_VEL
LIN {X 0,Y 372.229,Z 1053.74,A -85,B 0,C 180,E1 15622.621,E2 15622.621} C_VEL
LIN {X 0,Y 381.686,Z 1051.265,A -85,B 0,C 180,E1 15621.237,E2 15621.237} C_VEL
LIN {X 0,Y 395.769,Z 1046.964,A -85,B 0,C 180,E1 15619.511,E2 15619.511} C_VEL
LIN {X 0,Y 397.968,Z 1046.218,A -85,B 0,C 180,E1 15619.275,E2 15619.275} C_VEL
LIN {X 0,Y 389.463,Z 1064.523,A -85,B 0,C 180,E1 15616.601,E2 15616.601} C_VEL
LIN {X 0,Y 381.166,Z 1082.183,A -85,B 0,C 180,E1 15613.613,E2 15613.613} C_VEL
LIN {X 0,Y 373.413,Z 1098.307,A -85,B 0,C 180,E1 15610.393,E2 15610.393} C_VEL
LIN {X 0,Y 366.307,Z 1113.429,A -85,B 0,C 180,E1 15606.89,E2 15606.89} C_VEL
LIN {X 0,Y 360.358,Z 1126.392,A -85,B 0,C 180,E1 15603.327,E2 15603.327} C_VEL
LIN {X 0,Y 355.249,Z 1138.382,A -85,B 0,C 180,E1 15599.511,E2 15599.511} C_VEL
LIN {X 0,Y 351.092,Z 1148.88,A -85,B 0,C 180,E1 15595.471,E2 15595.471} C_VEL
LIN {X 0,Y 348.378,Z 1156.734,A -85,B 0,C 180,E1 15591.91,E2 15591.91} C_VEL
LIN {X 0,Y 346.088,Z 1164.723,A -85,B 0,C 180,E1 15587.488,E2 15587.488} C_VEL
LIN {X 0,Y 344.919,Z 1169.978,A -85,B 0,C 180,E1 15583.753,E2 15583.753} C_VEL
LIN {X 0,Y 344.344,Z 1173.678,A -85,B 0,C 180,E1 15580.374,E2 15580.374} C_VEL
LIN {X 0,Y 344.075,Z 1176.355,A -85,B 0,C 180,E1 15577.013,E2 15577.013} C_VEL
LIN {X 0,Y 343.981,Z 1178.229,A -85,B 0,C 180,E1 15573.168,E2 15573.168} C_VEL
LIN {X 0,Y 343.961,Z 1178.619,A -85,B 0,C 180,E1 15569.169,E2 15569.169} C_VEL
LIN {X 0,Y 343.99,Z 1177.851,A -85,B 0,C 180,E1 15565.835,E2 15565.835} C_VEL
LIN {X 0,Y 344.088,Z 1176.191,A -85,B 0,C 180,E1 15562.656,E2 15562.656} C_VEL
LIN {X 0,Y 344.354,Z 1173.611,A -85,B 0,C 180,E1 15559.462,E2 15559.462} C_VEL
LIN {X 0,Y 344.943,Z 1169.89,A -85,B 0,C 180,E1 15556.081,E2 15556.081} C_VEL
LIN {X 0,Y 346.261,Z 1164.108,A -85,B 0,C 180,E1 15552.005,E2 15552.005} C_VEL
LIN {X 0,Y 348.426,Z 1156.581,A -85,B 0,C 180,E1 15547.92,E2 15547.92} C_VEL
LIN {X 0,Y 351.017,Z 1149.109,A -85,B 0,C 180,E1 15544.527,E2 15544.527} C_VEL
LIN {X 0,Y 352.706,Z 1144.684,A -85,B 0,C 180,E1 15542.723,E2 15542.723} C_VEL
LIN {X 0,Y 352.924,Z 1141.824,A -85,B 0,C 180,E1 15541.556,E2 15541.556} C_VEL
LIN {X 0,Y 350.55,Z 1134.392,A -85,B 0,C 180,E1 15538.334,E2 15538.334} C_VEL
LIN {X 0,Y 351.173,Z 1131.651,A -85,B 0,C 180,E1 15537.342,E2 15537.342} C_VEL
LIN {X 0,Y 357.163,Z 1118.893,A -85,B 0,C 180,E1 15533.597,E2 15533.597} C_VEL
LIN {X 0,Y 363.444,Z 1106.061,A -85,B 0,C 180,E1 15530.341,E2 15530.341} C_VEL
LIN {X 0,Y 371.515,Z 1089.849,A -85,B 0,C 180,E1 15526.834,E2 15526.834} C_VEL
LIN {X 0,Y 378.789,Z 1075.216,A -85,B 0,C 180,E1 15524.114,E2 15524.114} C_VEL
LIN {X 0,Y 387.805,Z 1056.804,A -85,B 0,C 180,E1 15521.164,E2 15521.164} C_VEL
LIN {X 0,Y 395.906,Z 1039.585,A -85,B 0,C 180,E1 15518.811,E2 15518.811} C_VEL
LIN {X 0,Y 405.068,Z 1019.372,A -85,B 0,C 180,E1 15516.422,E2 15516.422} C_VEL
LIN {X 0,Y 413.107,Z 1000.239,A -85,B 0,C 180,E1 15514.498,E2 15514.498} C_VEL
LIN {X 0,Y 421.563,Z 979.053,A -85,B 0,C 180,E1 15512.651,E2 15512.651} C_VEL
LIN {X 0,Y 429.423,Z 957.045,A -85,B 0,C 180,E1 15511.038,E2 15511.038} C_VEL
LIN {X 0,Y 436.958,Z 934.108,A -85,B 0,C 180,E1 15509.598,E2 15509.598} C_VEL
LIN {X 0,Y 443.698,Z 910.265,A -85,B 0,C 180,E1 15508.362,E2 15508.362} C_VEL
LIN {X 0,Y 449.794,Z 885.812,A -85,B 0,C 180,E1 15507.302,E2 15507.302} C_VEL
LIN {X 0,Y 454.832,Z 860.979,A -85,B 0,C 180,E1 15506.442,E2 15506.442} C_VEL
LIN {X 0,Y 462.41,Z 818.594,A -85,B 0,C 180,E1 15505.29,E2 15505.29} C_VEL
LIN {X 0,Y 475.208,Z 744.366,A -85,B 0,C 180,E1 15503.59,E2 15503.59} C_VEL
LIN {X 0,Y 486.026,Z 673.632,A -85,B 0,C 180,E1 15502.152,E2 15502.152} C_VEL
LIN {X 0,Y 494.66,Z 607.388,A -85,B 0,C 180,E1 15500.944,E2 15500.944} C_VEL
LIN {X 0,Y 499.215,Z 565.434,A -85,B 0,C 180,E1 15500.213,E2 15500.213} C_VEL
LIN {X 0,Y 491.996,Z 559.967,A -85,B 0,C 180,E1 15497.383,E2 15497.383} C_VEL
LIN {X 0,Y 484.551,Z 556.546,A -85,B 0,C 180,E1 15493.971,E2 15493.971} C_VEL
LIN {X 0,Y 478.219,Z 554.816,A -85,B 0,C 180,E1 15490.237,E2 15490.237} C_VEL
LIN {X 0,Y 476.885,Z 554.932,A -85,B 0,C 180,E1 15489.291,E2 15489.291} C_VEL
LIN {X 0,Y 472.766,Z 556.823,A -85,B 0,C 180,E1 15485.583,E2 15485.583} C_VEL
LIN {X 0,Y 470.729,Z 560.111,A -85,B 0,C 180,E1 15482.678,E2 15482.678} C_VEL
LIN {X 0,Y 469.686,Z 565.456,A -85,B 0,C 180,E1 15479.39,E2 15479.39} C_VEL
LIN {X 0,Y 470.097,Z 574.418,A -85,B 0,C 180,E1 15475.547,E2 15475.547} C_VEL
LIN {X 0,Y 470.434,Z 577.034,A -85,B 0,C 180,E1 15474.649,E2 15474.649} C_VEL
LIN {X 0,Y 468.873,Z 609.689,A -85,B 0,C 180,E1 15472.132,E2 15472.132} C_VEL
LIN {X 0,Y 467.958,Z 642.048,A -85,B 0,C 180,E1 15469.816,E2 15469.816} C_VEL
LIN {X 0,Y 467.434,Z 681.412,A -85,B 0,C 180,E1 15467.067,E2 15467.067} C_VEL
LIN {X 0,Y 467.824,Z 705.196,A -85,B 0,C 180,E1 15465.17,E2 15465.17} C_VEL
LIN {X 0,Y 468.978,Z 728.381,A -85,B 0,C 180,E1 15463.112,E2 15463.112} C_VEL
LIN {X 0,Y 471.302,Z 751.112,A -85,B 0,C 180,E1 15460.818,E2 15460.818} C_VEL
LIN {X 0,Y 474.492,Z 770.565,A -85,B 0,C 180,E1 15458.641,E2 15458.641} C_VEL
LIN {X 0,Y 478.645,Z 788.708,A -85,B 0,C 180,E1 15456.447,E2 15456.447} C_VEL
LIN {X 0,Y 471.408,Z 828.797,A -85,B 0,C 180,E1 15455.562,E2 15455.562} C_VEL
LIN {X 0,Y 463.087,Z 867.298,A -85,B 0,C 180,E1 15454.569,E2 15454.569} C_VEL
LIN {X 0,Y 454.95,Z 901.46,A -85,B 0,C 180,E1 15453.44,E2 15453.44} C_VEL
LIN {X 0,Y 446.522,Z 934.111,A -85,B 0,C 180,E1 15452.095,E2 15452.095} C_VEL
LIN {X 0,Y 438.024,Z 965.084,A -85,B 0,C 180,E1 15450.554,E2 15450.554} C_VEL
LIN {X 0,Y 430.653,Z 990.228,A -85,B 0,C 180,E1 15449.077,E2 15449.077} C_VEL
LIN {X 0,Y 423.188,Z 1012.316,A -85,B 0,C 180,E1 15447.507,E2 15447.507} C_VEL
LIN {X 0,Y 415.466,Z 1032.726,A -85,B 0,C 180,E1 15445.787,E2 15445.787} C_VEL
LIN {X 0,Y 407.815,Z 1051.418,A -85,B 0,C 180,E1 15443.954,E2 15443.954} C_VEL
LIN {X 0,Y 399.221,Z 1070.483,A -85,B 0,C 180,E1 15441.735,E2 15441.735} C_VEL
LIN {X 0,Y 390.334,Z 1088.827,A -85,B 0,C 180,E1 15439.215,E2 15439.215} C_VEL
LIN {X 0,Y 381.767,Z 1105.613,A -85,B 0,C 180,E1 15436.506,E2 15436.506} C_VEL
LIN {X 0,Y 372.928,Z 1122.082,A -85,B 0,C 180,E1 15433.341,E2 15433.341} C_VEL
LIN {X 0,Y 364.687,Z 1136.923,A -85,B 0,C 180,E1 15429.906,E2 15429.906} C_VEL
LIN {X 0,Y 357.478,Z 1149.809,A -85,B 0,C 180,E1 15426.336,E2 15426.336} C_VEL
LIN {X 0,Y 350.949,Z 1161.678,A -85,B 0,C 180,E1 15422.384,E2 15422.384} C_VEL
LIN {X 0,Y 345.522,Z 1172.123,A -85,B 0,C 180,E1 15418.142,E2 15418.142} C_VEL
LIN {X 0,Y 341.477,Z 1180.739,A -85,B 0,C 180,E1 15413.831,E2 15413.831} C_VEL
LIN {X 0,Y 338.604,Z 1187.923,A -85,B 0,C 180,E1 15409.311,E2 15409.311} C_VEL
LIN {X 0,Y 336.942,Z 1193.43,A -85,B 0,C 180,E1 15404.784,E2 15404.784} C_VEL
LIN {X 0,Y 336.19,Z 1197.229,A -85,B 0,C 180,E1 15400.45,E2 15400.45} C_VEL
LIN {X 0,Y 335.979,Z 1199.64,A -85,B 0,C 180,E1 15396.276,E2 15396.276} C_VEL
LIN {X 0,Y 335.964,Z 1200.859,A -85,B 0,C 180,E1 15392.215,E2 15392.215} C_VEL
LIN {X 0,Y 335.97,Z 1200.917,A -85,B 0,C 180,E1 15388.463,E2 15388.463} C_VEL
LIN {X 0,Y 335.968,Z 1199.98,A -85,B 0,C 180,E1 15384.533,E2 15384.533} C_VEL
LIN {X 0,Y 336.104,Z 1197.957,A -85,B 0,C 180,E1 15380.581,E2 15380.581} C_VEL
LIN {X 0,Y 336.705,Z 1194.369,A -85,B 0,C 180,E1 15376.186,E2 15376.186} C_VEL
LIN {X 0,Y 338.204,Z 1189.061,A -85,B 0,C 180,E1 15371.556,E2 15371.556} C_VEL
LIN {X 0,Y 340.951,Z 1181.918,A -85,B 0,C 180,E1 15366.858,E2 15366.858} C_VEL
LIN {X 0,Y 344.969,Z 1173.224,A -85,B 0,C 180,E1 15362.368,E2 15362.368} C_VEL
LIN {X 0,Y 350.239,Z 1163.019,A -85,B 0,C 180,E1 15358.118,E2 15358.118} C_VEL
LIN {X 0,Y 356.631,Z 1151.317,A -85,B 0,C 180,E1 15354.123,E2 15354.123} C_VEL
LIN {X 0,Y 364.004,Z 1138.163,A -85,B 0,C 180,E1 15350.409,E2 15350.409} C_VEL
LIN {X 0,Y 372.15,Z 1123.409,A -85,B 0,C 180,E1 15346.954,E2 15346.954} C_VEL
LIN {X 0,Y 380.439,Z 1108.004,A -85,B 0,C 180,E1 15343.932,E2 15343.932} C_VEL
LIN {X 0,Y 389.572,Z 1090.327,A -85,B 0,C 180,E1 15341.009,E2 15341.009} C_VEL
LIN {X 0,Y 398.715,Z 1071.521,A -85,B 0,C 180,E1 15338.399,E2 15338.399} C_VEL
LIN {X 0,Y 407.766,Z 1051.384,A -85,B 0,C 180,E1 15336.051,E2 15336.051} C_VEL
LIN {X 0,Y 416.256,Z 1030.693,A -85,B 0,C 180,E1 15334.03,E2 15334.03} C_VEL
LIN {X 0,Y 424.373,Z 1008.785,A -85,B 0,C 180,E1 15332.234,E2 15332.234} C_VEL
LIN {X 0,Y 431.866,Z 985.986,A -85,B 0,C 180,E1 15330.668,E2 15330.668} C_VEL
LIN {X 0,Y 440.879,Z 954.734,A -85,B 0,C 180,E1 15328.903,E2 15328.903} C_VEL
LIN {X 0,Y 450.111,Z 920.194,A -85,B 0,C 180,E1 15327.304,E2 15327.304} C_VEL
LIN {X 0,Y 458.505,Z 886.468,A -85,B 0,C 180,E1 15326.04,E2 15326.04} C_VEL
LIN {X 0,Y 466.725,Z 850.714,A -85,B 0,C 180,E1 15324.981,E2 15324.981} C_VEL
LIN {X 0,Y 474.828,Z 810.359,A -85,B 0,C 180,E1 15324.021,E2 15324.021} C_VEL
LIN {X 0,Y 481.676,Z 768.146,A -85,B 0,C 180,E1 15323.159,E2 15323.159} C_VEL
LIN {X 0,Y 487.345,Z 723.662,A -85,B 0,C 180,E1 15322.423,E2 15322.423} C_VEL
LIN {X 0,Y 491.876,Z 674.615,A -85,B 0,C 180,E1 15321.76,E2 15321.76} C_VEL
LIN {X 0,Y 492.472,Z 667.847,A -85,B 0,C 180,E1 15321.679,E2 15321.679} C_VEL
LIN {X 0,Y 485.668,Z 691.878,A -85,B 0,C 180,E1 15320.582,E2 15320.582} C_VEL
LIN {X 0,Y 480.624,Z 707.751,A -85,B 0,C 180,E1 15319.72,E2 15319.72} C_VEL
LIN {X 0,Y 473.977,Z 729.385,A -85,B 0,C 180,E1 15318.743,E2 15318.743} C_VEL
LIN {X 0,Y 467.19,Z 748.263,A -85,B 0,C 180,E1 15317.677,E2 15317.677} C_VEL
LIN {X 0,Y 460.302,Z 767.685,A -85,B 0,C 180,E1 15316.725,E2 15316.725} C_VEL
LIN {X 0,Y 454.438,Z 782.35,A -85,B 0,C 180,E1 15315.824,E2 15315.824} C_VEL
LIN {X 0,Y 447.612,Z 799.91,A -85,B 0,C 180,E1 15314.886,E2 15314.886} C_VEL
LIN {X 0,Y 442.609,Z 811.603,A -85,B 0,C 180,E1 15314.113,E2 15314.113} C_VEL
LIN {X 0,Y 435.778,Z 828.082,A -85,B 0,C 180,E1 15313.163,E2 15313.163} C_VEL
LIN {X 0,Y 431.364,Z 837.977,A -85,B 0,C 180,E1 15312.466,E2 15312.466} C_VEL
LIN {X 0,Y 424.836,Z 853.173,A -85,B 0,C 180,E1 15311.529,E2 15311.529} C_VEL
LIN {X 0,Y 420.635,Z 862.417,A -85,B 0,C 180,E1 15310.841,E2 15310.841} C_VEL
LIN {X 0,Y 414.515,Z 876.304,A -85,B 0,C 180,E1 15309.932,E2 15309.932} C_VEL
LIN {X 0,Y 411.297,Z 883.182,A -85,B 0,C 180,E1 15309.374,E2 15309.374} C_VEL
LIN {X 0,Y 404.624,Z 898.609,A -85,B 0,C 180,E1 15308.448,E2 15308.448} C_VEL
LIN {X 0,Y 401.903,Z 904.619,A -85,B 0,C 180,E1 15308.03,E2 15308.03} C_VEL
LIN {X 0,Y 396.62,Z 917.184,A -85,B 0,C 180,E1 15307.486,E2 15307.486} C_VEL
LIN {X 0,Y 393.441,Z 924.488,A -85,B 0,C 180,E1 15307.054,E2 15307.054} C_VEL
LIN {X 0,Y 388.081,Z 936.651,A -85,B 0,C 180,E1 15306.509,E2 15306.509} C_VEL
LIN {X 0,Y 384.052,Z 944.935,A -85,B 0,C 180,E1 15305.977,E2 15305.977} C_VEL
LIN {X 0,Y 379.115,Z 954.833,A -85,B 0,C 180,E1 15305.448,E2 15305.448} C_VEL
LIN {X 0,Y 375.949,Z 960.515,A -85,B 0,C 180,E1 15305.006,E2 15305.006} C_VEL
LIN {X 0,Y 371.696,Z 968.256,A -85,B 0,C 180,E1 15304.552,E2 15304.552} C_VEL
LIN {X 0,Y 367.863,Z 974.625,A -85,B 0,C 180,E1 15304.001,E2 15304.001} C_VEL
LIN {X 0,Y 363.503,Z 981.789,A -85,B 0,C 180,E1 15303.469,E2 15303.469} C_VEL
LIN {X 0,Y 360.927,Z 985.744,A -85,B 0,C 180,E1 15303.047,E2 15303.047} C_VEL
LIN {X 0,Y 357.128,Z 991.565,A -85,B 0,C 180,E1 15302.568,E2 15302.568} C_VEL
LIN {X 0,Y 354.868,Z 994.836,A -85,B 0,C 180,E1 15302.133,E2 15302.133} C_VEL
LIN {X 0,Y 351.553,Z 999.75,A -85,B 0,C 180,E1 15301.711,E2 15301.711} C_VEL
LIN {X 0,Y 349.628,Z 1002.539,A -85,B 0,C 180,E1 15301.219,E2 15301.219} C_VEL
LIN {X 0,Y 349.399,Z 1019.371,A -85,B 0,C 180,E1 15300.533,E2 15300.533} C_VEL
LIN {X 0,Y 348.9,Z 1032.344,A -85,B 0,C 180,E1 15299.754,E2 15299.754} C_VEL
LIN {X 0,Y 348.066,Z 1046.121,A -85,B 0,C 180,E1 15298.646,E2 15298.646} C_VEL
LIN {X 0,Y 347.022,Z 1058.13,A -85,B 0,C 180,E1 15297.358,E2 15297.358} C_VEL
LIN {X 0,Y 345.957,Z 1068.128,A -85,B 0,C 180,E1 15296.022,E2 15296.022} C_VEL
LIN {X 0,Y 344.669,Z 1078.291,A -85,B 0,C 180,E1 15294.307,E2 15294.307} C_VEL
LIN {X 0,Y 343.505,Z 1085.874,A -85,B 0,C 180,E1 15292.641,E2 15292.641} C_VEL
LIN {X 0,Y 342.45,Z 1092.022,A -85,B 0,C 180,E1 15290.928,E2 15290.928} C_VEL
LIN {X 0,Y 341.543,Z 1096.79,A -85,B 0,C 180,E1 15289.201,E2 15289.201} C_VEL
LIN {X 0,Y 340.733,Z 1100.668,A -85,B 0,C 180,E1 15287.286,E2 15287.286} C_VEL
LIN {X 0,Y 339.954,Z 1103.587,A -85,B 0,C 180,E1 15284.825,E2 15284.825} C_VEL
LIN {X 0,Y 339.511,Z 1104.353,A -85,B 0,C 180,E1 15282.695,E2 15282.695} C_VEL
LIN {X 0,Y 339.289,Z 1103.745,A -85,B 0,C 180,E1 15280.727,E2 15280.727} C_VEL
LIN {X 0,Y 339.253,Z 1101.736,A -85,B 0,C 180,E1 15278.651,E2 15278.651} C_VEL
LIN {X 0,Y 339.45,Z 1097.434,A -85,B 0,C 180,E1 15276.2,E2 15276.2} C_VEL
LIN {X 0,Y 339.81,Z 1092.264,A -85,B 0,C 180,E1 15274.214,E2 15274.214} C_VEL
LIN {X 0,Y 340.274,Z 1086.593,A -85,B 0,C 180,E1 15272.526,E2 15272.526} C_VEL
LIN {X 0,Y 340.951,Z 1078.823,A -85,B 0,C 180,E1 15270.676,E2 15270.676} C_VEL
LIN {X 0,Y 341.8,Z 1068.884,A -85,B 0,C 180,E1 15268.816,E2 15268.816} C_VEL
LIN {X 0,Y 342.382,Z 1062.23,A -85,B 0,C 180,E1 15267.744,E2 15267.744} C_VEL
LIN {X 0,Y 344.106,Z 1062.66,A -85,B 0,C 180,E1 15267.086,E2 15267.086} C_VEL
LIN {X 0,Y 345.845,Z 1062.408,A -85,B 0,C 180,E1 15266.675,E2 15266.675} C_VEL
LIN {X 0,Y 348.979,Z 1062.33,A -85,B 0,C 180,E1 15265.835,E2 15265.835} C_VEL
LIN {X 0,Y 358.491,Z 1061.16,A -85,B 0,C 180,E1 15263.75,E2 15263.75} C_VEL
LIN {X 0,Y 369.104,Z 1059.202,A -85,B 0,C 180,E1 15261.855,E2 15261.855} C_VEL
LIN {X 0,Y 378.697,Z 1056.764,A -85,B 0,C 180,E1 15260.482,E2 15260.482} C_VEL
LIN {X 0,Y 389.164,Z 1053.829,A -85,B 0,C 180,E1 15259.164,E2 15259.164} C_VEL
LIN {X 0,Y 379.838,Z 1073.053,A -85,B 0,C 180,E1 15256.162,E2 15256.162} C_VEL
LIN {X 0,Y 371.604,Z 1089.615,A -85,B 0,C 180,E1 15253.115,E2 15253.115} C_VEL
LIN {X 0,Y 363.261,Z 1106.38,A -85,B 0,C 180,E1 15249.484,E2 15249.484} C_VEL
LIN {X 0,Y 356.714,Z 1119.788,A -85,B 0,C 180,E1 15246.063,E2 15246.063} C_VEL
LIN {X 0,Y 350.231,Z 1133.639,A -85,B 0,C 180,E1 15241.883,E2 15241.883} C_VEL
LIN {X 0,Y 345.851,Z 1143.652,A -85,B 0,C 180,E1 15238.305,E2 15238.305} C_VEL
LIN {X 0,Y 341.884,Z 1153.851,A -85,B 0,C 180,E1 15233.989,E2 15233.989} C_VEL
LIN {X 0,Y 339.26,Z 1161.51,A -85,B 0,C 180,E1 15229.993,E2 15229.993} C_VEL
LIN {X 0,Y 337.68,Z 1167.284,A -85,B 0,C 180,E1 15226.34,E2 15226.34} C_VEL
LIN {X 0,Y 336.584,Z 1172.656,A -85,B 0,C 180,E1 15222.004,E2 15222.004} C_VEL
LIN {X 0,Y 336.16,Z 1175.927,A -85,B 0,C 180,E1 15218.21,E2 15218.21} C_VEL
LIN {X 0,Y 336.009,Z 1177.798,A -85,B 0,C 180,E1 15214.953,E2 15214.953} C_VEL
LIN {X 0,Y 335.971,Z 1178.752,A -85,B 0,C 180,E1 15211.708,E2 15211.708} C_VEL
LIN {X 0,Y 335.971,Z 1178.811,A -85,B 0,C 180,E1 15208.638,E2 15208.638} C_VEL
LIN {X 0,Y 336,Z 1177.975,A -85,B 0,C 180,E1 15205.394,E2 15205.394} C_VEL
LIN {X 0,Y 336.128,Z 1176.222,A -85,B 0,C 180,E1 15202.135,E2 15202.135} C_VEL
LIN {X 0,Y 336.464,Z 1173.39,A -85,B 0,C 180,E1 15198.691,E2 15198.691} C_VEL
LIN {X 0,Y 337.42,Z 1168.49,A -85,B 0,C 180,E1 15194.385,E2 15194.385} C_VEL
LIN {X 0,Y 339.035,Z 1162.284,A -85,B 0,C 180,E1 15190.356,E2 15190.356} C_VEL
LIN {X 0,Y 341.287,Z 1155.444,A -85,B 0,C 180,E1 15186.704,E2 15186.704} C_VEL
LIN {X 0,Y 344.992,Z 1145.844,A -85,B 0,C 180,E1 15182.432,E2 15182.432} C_VEL
LIN {X 0,Y 349.428,Z 1135.422,A -85,B 0,C 180,E1 15178.617,E2 15178.617} C_VEL
LIN {X 0,Y 351.173,Z 1131.651,A -85,B 0,C 180,E1 15177.342,E2 15177.342} C_VEL
LIN {X 0,Y 351.869,Z 1128.426,A -85,B 0,C 180,E1 15176.196,E2 15176.196} C_VEL
LIN {X 0,Y 350.773,Z 1119.8,A -85,B 0,C 180,E1 15173.034,E2 15173.034} C_VEL
LIN {X 0,Y 351.757,Z 1116.658,A -85,B 0,C 180,E1 15172.088,E2 15172.088} C_VEL
LIN {X 0,Y 359.977,Z 1100.78,A -85,B 0,C 180,E1 15168.195,E2 15168.195} C_VEL
LIN {X 0,Y 367.458,Z 1086.393,A -85,B 0,C 180,E1 15165.193,E2 15165.193} C_VEL
LIN {X 0,Y 376.736,Z 1068.346,A -85,B 0,C 180,E1 15161.977,E2 15161.977} C_VEL
LIN {X 0,Y 385.015,Z 1051.801,A -85,B 0,C 180,E1 15159.457,E2 15159.457} C_VEL
LIN {X 0,Y 394.982,Z 1031.012,A -85,B 0,C 180,E1 15156.758,E2 15156.758} C_VEL
LIN {X 0,Y 403.593,Z 1012.07,A -85,B 0,C 180,E1 15154.667,E2 15154.667} C_VEL
LIN {X 0,Y 413.285,Z 989.108,A -85,B 0,C 180,E1 15152.517,E2 15152.517} C_VEL
LIN {X 0,Y 421.518,Z 967.924,A -85,B 0,C 180,E1 15150.833,E2 15150.833} C_VEL
LIN {X 0,Y 429.436,Z 945.232,A -85,B 0,C 180,E1 15149.316,E2 15149.316} C_VEL
LIN {X 0,Y 435.944,Z 924.553,A -85,B 0,C 180,E1 15148.133,E2 15148.133} C_VEL
LIN {X 0,Y 442.93,Z 899.023,A -85,B 0,C 180,E1 15146.919,E2 15146.919} C_VEL
LIN {X 0,Y 447.851,Z 877.973,A -85,B 0,C 180,E1 15146.093,E2 15146.093} C_VEL
LIN {X 0,Y 453.378,Z 849.581,A -85,B 0,C 180,E1 15145.19,E2 15145.19} C_VEL
LIN {X 0,Y 464.009,Z 791.615,A -85,B 0,C 180,E1 15143.745,E2 15143.745} C_VEL
LIN {X 0,Y 476.181,Z 719.815,A -85,B 0,C 180,E1 15142.174,E2 15142.174} C_VEL
LIN {X 0,Y 486.211,Z 652.363,A -85,B 0,C 180,E1 15140.862,E2 15140.862} C_VEL
LIN {X 0,Y 494.194,Z 588.424,A -85,B 0,C 180,E1 15139.74,E2 15139.74} C_VEL
LIN {X 0,Y 495.942,Z 572.061,A -85,B 0,C 180,E1 15139.461,E2 15139.461} C_VEL
LIN {X 0,Y 490.399,Z 567.71,A -85,B 0,C 180,E1 15137.196,E2 15137.196} C_VEL
LIN {X 0,Y 483.326,Z 564.438,A -85,B 0,C 180,E1 15133.885,E2 15133.885} C_VEL
LIN {X 0,Y 477.081,Z 562.721,A -85,B 0,C 180,E1 15130.14,E2 15130.14} C_VEL
LIN {X 0,Y 475.585,Z 563.028,A -85,B 0,C 180,E1 15129.073,E2 15129.073} C_VEL
LIN {X 0,Y 471.895,Z 564.705,A -85,B 0,C 180,E1 15125.715,E2 15125.715} C_VEL
LIN {X 0,Y 469.873,Z 567.815,A -85,B 0,C 180,E1 15122.928,E2 15122.928} C_VEL
LIN {X 0,Y 468.718,Z 573.143,A -85,B 0,C 180,E1 15119.633,E2 15119.633} C_VEL
LIN {X 0,Y 469.019,Z 582.26,A -85,B 0,C 180,E1 15115.721,E2 15115.721} C_VEL
LIN {X 0,Y 469.14,Z 583.704,A -85,B 0,C 180,E1 15115.278,E2 15115.278} C_VEL
LIN {X 0,Y 467.421,Z 614.667,A -85,B 0,C 180,E1 15112.893,E2 15112.893} C_VEL
LIN {X 0,Y 466.138,Z 650.168,A -85,B 0,C 180,E1 15110.345,E2 15110.345} C_VEL
LIN {X 0,Y 465.323,Z 683.255,A -85,B 0,C 180,E1 15108.032,E2 15108.032} C_VEL
LIN {X 0,Y 465.332,Z 707.761,A -85,B 0,C 180,E1 15106.09,E2 15106.09} C_VEL
LIN {X 0,Y 466.122,Z 731.466,A -85,B 0,C 180,E1 15103.983,E2 15103.983} C_VEL
LIN {X 0,Y 468.147,Z 755.432,A -85,B 0,C 180,E1 15101.556,E2 15101.556} C_VEL
LIN {X 0,Y 471.15,Z 775.88,A -85,B 0,C 180,E1 15099.242,E2 15099.242} C_VEL
LIN {X 0,Y 474.577,Z 792.269,A -85,B 0,C 180,E1 15097.245,E2 15097.245} C_VEL
LIN {X 0,Y 466.481,Z 835.204,A -85,B 0,C 180,E1 15096.285,E2 15096.285} C_VEL
LIN {X 0,Y 458.098,Z 872.169,A -85,B 0,C 180,E1 15095.3,E2 15095.3} C_VEL
LIN {X 0,Y 449.524,Z 906.912,A -85,B 0,C 180,E1 15094.119,E2 15094.119} C_VEL
LIN {X 0,Y 440.894,Z 939.533,A -85,B 0,C 180,E1 15092.743,E2 15092.743} C_VEL
LIN {X 0,Y 432.064,Z 970.671,A -85,B 0,C 180,E1 15091.15,E2 15091.15} C_VEL
LIN {X 0,Y 424.983,Z 993.348,A -85,B 0,C 180,E1 15089.768,E2 15089.768} C_VEL
LIN {X 0,Y 417.751,Z 1014.127,A -85,B 0,C 180,E1 15088.271,E2 15088.271} C_VEL
LIN {X 0,Y 409.544,Z 1034.949,A -85,B 0,C 180,E1 15086.483,E2 15086.483} C_VEL
LIN {X 0,Y 401.005,Z 1054.602,A -85,B 0,C 180,E1 15084.481,E2 15084.481} C_VEL
LIN {X 0,Y 392.558,Z 1072.798,A -85,B 0,C 180,E1 15082.316,E2 15082.316} C_VEL
LIN {X 0,Y 383.556,Z 1090.641,A -85,B 0,C 180,E1 15079.798,E2 15079.798} C_VEL
LIN {X 0,Y 374.589,Z 1107.373,A -85,B 0,C 180,E1 15076.999,E2 15076.999} C_VEL
LIN {X 0,Y 365.967,Z 1122.874,A -85,B 0,C 180,E1 15073.942,E2 15073.942} C_VEL
LIN {X 0,Y 357.549,Z 1137.556,A -85,B 0,C 180,E1 15070.478,E2 15070.478} C_VEL
LIN {X 0,Y 349.505,Z 1151.43,A -85,B 0,C 180,E1 15066.514,E2 15066.514} C_VEL
LIN {X 0,Y 342.857,Z 1163.061,A -85,B 0,C 180,E1 15062.45,E2 15062.45} C_VEL
LIN {X 0,Y 337.372,Z 1173.22,A -85,B 0,C 180,E1 15058.112,E2 15058.112} C_VEL
LIN {X 0,Y 333.176,Z 1181.87,A -85,B 0,C 180,E1 15053.522,E2 15053.522} C_VEL
LIN {X 0,Y 330.384,Z 1188.739,A -85,B 0,C 180,E1 15048.892,E2 15048.892} C_VEL
LIN {X 0,Y 328.803,Z 1193.972,A -85,B 0,C 180,E1 15044.257,E2 15044.257} C_VEL
LIN {X 0,Y 328.135,Z 1197.576,A -85,B 0,C 180,E1 15039.823,E2 15039.823} C_VEL
LIN {X 0,Y 327.976,Z 1199.642,A -85,B 0,C 180,E1 15035.772,E2 15035.772} C_VEL
LIN {X 0,Y 327.974,Z 1200.64,A -85,B 0,C 180,E1 15031.745,E2 15031.745} C_VEL
LIN {X 0,Y 327.969,Z 1200.609,A -85,B 0,C 180,E1 15027.901,E2 15027.901} C_VEL
LIN {X 0,Y 327.979,Z 1199.495,A -85,B 0,C 180,E1 15023.873,E2 15023.873} C_VEL
LIN {X 0,Y 328.18,Z 1197.206,A -85,B 0,C 180,E1 15019.642,E2 15019.642} C_VEL
LIN {X 0,Y 328.984,Z 1193.303,A -85,B 0,C 180,E1 15015.026,E2 15015.026} C_VEL
LIN {X 0,Y 330.725,Z 1187.806,A -85,B 0,C 180,E1 15010.39,E2 15010.39} C_VEL
LIN {X 0,Y 333.726,Z 1180.653,A -85,B 0,C 180,E1 15005.764,E2 15005.764} C_VEL
LIN {X 0,Y 338.152,Z 1171.695,A -85,B 0,C 180,E1 15001.183,E2 15001.183} C_VEL
LIN {X 0,Y 343.86,Z 1161.199,A -85,B 0,C 180,E1 14996.859,E2 14996.859} C_VEL
LIN {X 0,Y 350.752,Z 1149.193,A -85,B 0,C 180,E1 14992.816,E2 14992.816} C_VEL
LIN {X 0,Y 358.584,Z 1135.693,A -85,B 0,C 180,E1 14989.057,E2 14989.057} C_VEL
LIN {X 0,Y 367.226,Z 1120.674,A -85,B 0,C 180,E1 14985.59,E2 14985.59} C_VEL
LIN {X 0,Y 376.435,Z 1104.025,A -85,B 0,C 180,E1 14982.401,E2 14982.401} C_VEL
LIN {X 0,Y 385.533,Z 1086.696,A -85,B 0,C 180,E1 14979.62,E2 14979.62} C_VEL
LIN {X 0,Y 394.885,Z 1067.77,A -85,B 0,C 180,E1 14977.06,E2 14977.06} C_VEL
LIN {X 0,Y 404.113,Z 1047.595,A -85,B 0,C 180,E1 14974.767,E2 14974.767} C_VEL
LIN {X 0,Y 413.056,Z 1026.176,A -85,B 0,C 180,E1 14972.732,E2 14972.732} C_VEL
LIN {X 0,Y 421.472,Z 1003.625,A -85,B 0,C 180,E1 14970.949,E2 14970.949} C_VEL
LIN {X 0,Y 428.879,Z 981.142,A -85,B 0,C 180,E1 14969.467,E2 14969.467} C_VEL
LIN {X 0,Y 437.769,Z 950.526,A -85,B 0,C 180,E1 14967.793,E2 14967.793} C_VEL
LIN {X 0,Y 447.068,Z 916.22,A -85,B 0,C 180,E1 14966.251,E2 14966.251} C_VEL
LIN {X 0,Y 455.868,Z 881.2,A -85,B 0,C 180,E1 14964.984,E2 14964.984} C_VEL
LIN {X 0,Y 464.19,Z 845.27,A -85,B 0,C 180,E1 14963.969,E2 14963.969} C_VEL
LIN {X 0,Y 472.293,Z 804.7,A -85,B 0,C 180,E1 14963.026,E2 14963.026} C_VEL
LIN {X 0,Y 478.989,Z 763.614,A -85,B 0,C 180,E1 14962.208,E2 14962.208} C_VEL
LIN {X 0,Y 484.551,Z 720.712,A -85,B 0,C 180,E1 14961.513,E2 14961.513} C_VEL
LIN {X 0,Y 486.648,Z 699.285,A -85,B 0,C 180,E1 14961.184,E2 14961.184} C_VEL
LIN {X 0,Y 482.685,Z 711.408,A -85,B 0,C 180,E1 14960.534,E2 14960.534} C_VEL
LIN {X 0,Y 475.809,Z 733.256,A -85,B 0,C 180,E1 14959.56,E2 14959.56} C_VEL
LIN {X 0,Y 468.958,Z 751.923,A -85,B 0,C 180,E1 14958.523,E2 14958.523} C_VEL
LIN {X 0,Y 461.847,Z 771.487,A -85,B 0,C 180,E1 14957.579,E2 14957.579} C_VEL
LIN {X 0,Y 455.816,Z 786.249,A -85,B 0,C 180,E1 14956.692,E2 14956.692} C_VEL
LIN {X 0,Y 448.751,Z 803.946,A -85,B 0,C 180,E1 14955.757,E2 14955.757} C_VEL
LIN {X 0,Y 443.704,Z 815.469,A -85,B 0,C 180,E1 14955.012,E2 14955.012} C_VEL
LIN {X 0,Y 436.594,Z 832.193,A -85,B 0,C 180,E1 14954.059,E2 14954.059} C_VEL
LIN {X 0,Y 432.125,Z 841.951,A -85,B 0,C 180,E1 14953.388,E2 14953.388} C_VEL
LIN {X 0,Y 425.269,Z 857.386,A -85,B 0,C 180,E1 14952.445,E2 14952.445} C_VEL
LIN {X 0,Y 421.485,Z 865.465,A -85,B 0,C 180,E1 14951.842,E2 14951.842} C_VEL
LIN {X 0,Y 414.881,Z 880.076,A -85,B 0,C 180,E1 14950.906,E2 14950.906} C_VEL
LIN {X 0,Y 411.503,Z 887.08,A -85,B 0,C 180,E1 14950.359,E2 14950.359} C_VEL
LIN {X 0,Y 404.322,Z 903.137,A -85,B 0,C 180,E1 14949.394,E2 14949.394} C_VEL
LIN {X 0,Y 402.353,Z 907.351,A -85,B 0,C 180,E1 14949.105,E2 14949.105} C_VEL
LIN {X 0,Y 396.82,Z 920.31,A -85,B 0,C 180,E1 14948.55,E2 14948.55} C_VEL
LIN {X 0,Y 393.421,Z 927.867,A -85,B 0,C 180,E1 14948.134,E2 14948.134} C_VEL
LIN {X 0,Y 387.701,Z 940.443,A -85,B 0,C 180,E1 14947.558,E2 14947.558} C_VEL
LIN {X 0,Y 383.905,Z 947.835,A -85,B 0,C 180,E1 14947.097,E2 14947.097} C_VEL
LIN {X 0,Y 378.919,Z 957.508,A -85,B 0,C 180,E1 14946.591,E2 14946.591} C_VEL
LIN {X 0,Y 375.095,Z 964.291,A -85,B 0,C 180,E1 14946.108,E2 14946.108} C_VEL
LIN {X 0,Y 370.223,Z 972.688,A -85,B 0,C 180,E1 14945.58,E2 14945.58} C_VEL
LIN {X 0,Y 367.158,Z 977.657,A -85,B 0,C 180,E1 14945.156,E2 14945.156} C_VEL
LIN {X 0,Y 362.33,Z 985.288,A -85,B 0,C 180,E1 14944.59,E2 14944.59} C_VEL
LIN {X 0,Y 359.941,Z 988.83,A -85,B 0,C 180,E1 14944.217,E2 14944.217} C_VEL
LIN {X 0,Y 355.707,Z 995.141,A -85,B 0,C 180,E1 14943.696,E2 14943.696} C_VEL
LIN {X 0,Y 352.908,Z 999.065,A -85,B 0,C 180,E1 14943.248,E2 14943.248} C_VEL
LIN {X 0,Y 349.374,Z 1003.991,A -85,B 0,C 180,E1 14942.763,E2 14942.763} C_VEL
LIN {X 0,Y 347.264,Z 1006.779,A -85,B 0,C 180,E1 14942.364,E2 14942.364} C_VEL
LIN {X 0,Y 344.161,Z 1011.003,A -85,B 0,C 180,E1 14941.913,E2 14941.913} C_VEL
LIN {X 0,Y 342.421,Z 1013.4,A -85,B 0,C 180,E1 14941.438,E2 14941.438} C_VEL
LIN {X 0,Y 341.992,Z 1028.37,A -85,B 0,C 180,E1 14940.658,E2 14940.658} C_VEL
LIN {X 0,Y 341.186,Z 1041.667,A -85,B 0,C 180,E1 14939.664,E2 14939.664} C_VEL
LIN {X 0,Y 340.292,Z 1053.126,A -85,B 0,C 180,E1 14938.569,E2 14938.569} C_VEL
LIN {X 0,Y 338.926,Z 1066.108,A -85,B 0,C 180,E1 14936.956,E2 14936.956} C_VEL
LIN {X 0,Y 337.802,Z 1074.755,A -85,B 0,C 180,E1 14935.586,E2 14935.586} C_VEL
LIN {X 0,Y 336.718,Z 1082.162,A -85,B 0,C 180,E1 14934.16,E2 14934.16} C_VEL
LIN {X 0,Y 335.659,Z 1088.572,A -85,B 0,C 180,E1 14932.641,E2 14932.641} C_VEL
LIN {X 0,Y 334.573,Z 1094.444,A -85,B 0,C 180,E1 14930.886,E2 14930.886} C_VEL
LIN {X 0,Y 333.392,Z 1100.071,A -85,B 0,C 180,E1 14928.583,E2 14928.583} C_VEL
LIN {X 0,Y 332.527,Z 1103.371,A -85,B 0,C 180,E1 14926.435,E2 14926.435} C_VEL
LIN {X 0,Y 331.968,Z 1105.016,A -85,B 0,C 180,E1 14924.55,E2 14924.55} C_VEL
LIN {X 0,Y 331.582,Z 1105.503,A -85,B 0,C 180,E1 14922.63,E2 14922.63} C_VEL
LIN {X 0,Y 331.356,Z 1104.752,A -85,B 0,C 180,E1 14920.614,E2 14920.614} C_VEL
LIN {X 0,Y 331.333,Z 1102.215,A -85,B 0,C 180,E1 14918.211,E2 14918.211} C_VEL
LIN {X 0,Y 331.534,Z 1097.993,A -85,B 0,C 180,E1 14915.974,E2 14915.974} C_VEL
LIN {X 0,Y 331.886,Z 1093.119,A -85,B 0,C 180,E1 14914.097,E2 14914.097} C_VEL
LIN {X 0,Y 332.436,Z 1086.65,A -85,B 0,C 180,E1 14912.166,E2 14912.166} C_VEL
LIN {X 0,Y 333.302,Z 1076.906,A -85,B 0,C 180,E1 14909.934,E2 14909.934} C_VEL
LIN {X 0,Y 334.117,Z 1067.857,A -85,B 0,C 180,E1 14908.276,E2 14908.276} C_VEL
LIN {X 0,Y 335.787,Z 1068.331,A -85,B 0,C 180,E1 14907.588,E2 14907.588} C_VEL
LIN {X 0,Y 337.451,Z 1068.122,A -85,B 0,C 180,E1 14907.163,E2 14907.163} C_VEL
LIN {X 0,Y 340.474,Z 1068.117,A -85,B 0,C 180,E1 14906.286,E2 14906.286} C_VEL
LIN {X 0,Y 347.825,Z 1067.609,A -85,B 0,C 180,E1 14904.445,E2 14904.445} C_VEL
LIN {X 0,Y 359.038,Z 1065.967,A -85,B 0,C 180,E1 14902.216,E2 14902.216} C_VEL
LIN {X 0,Y 372.591,Z 1063.066,A -85,B 0,C 180,E1 14900.105,E2 14900.105} C_VEL
LIN {X 0,Y 380.39,Z 1061.096,A -85,B 0,C 180,E1 14899.082,E2 14899.082} C_VEL
LIN {X 0,Y 371.463,Z 1078.57,A -85,B 0,C 180,E1 14896.171,E2 14896.171} C_VEL
LIN {X 0,Y 362.026,Z 1096.782,A -85,B 0,C 180,E1 14892.586,E2 14892.586} C_VEL
LIN {X 0,Y 354.811,Z 1110.708,A -85,B 0,C 180,E1 14889.353,E2 14889.353} C_VEL
LIN {X 0,Y 347.081,Z 1125.888,A -85,B 0,C 180,E1 14885.184,E2 14885.184} C_VEL
LIN {X 0,Y 341.747,Z 1136.937,A -85,B 0,C 180,E1 14881.584,E2 14881.584} C_VEL
LIN {X 0,Y 336.525,Z 1148.649,A -85,B 0,C 180,E1 14877.041,E2 14877.041} C_VEL
LIN {X 0,Y 333.241,Z 1156.929,A -85,B 0,C 180,E1 14873.147,E2 14873.147} C_VEL
LIN {X 0,Y 330.648,Z 1164.766,A -85,B 0,C 180,E1 14868.698,E2 14868.698} C_VEL
LIN {X 0,Y 329.123,Z 1170.513,A -85,B 0,C 180,E1 14864.427,E2 14864.427} C_VEL
LIN {X 0,Y 328.433,Z 1174.209,A -85,B 0,C 180,E1 14860.882,E2 14860.882} C_VEL
LIN {X 0,Y 328.113,Z 1176.88,A -85,B 0,C 180,E1 14857.356,E2 14857.356} C_VEL
LIN {X 0,Y 327.995,Z 1178.683,A -85,B 0,C 180,E1 14853.498,E2 14853.498} C_VEL
LIN {X 0,Y 327.969,Z 1179.191,A -85,B 0,C 180,E1 14849.478,E2 14849.478} C_VEL
LIN {X 0,Y 328.001,Z 1178.445,A -85,B 0,C 180,E1 14845.807,E2 14845.807} C_VEL
LIN {X 0,Y 328.117,Z 1176.832,A -85,B 0,C 180,E1 14842.473,E2 14842.473} C_VEL
LIN {X 0,Y 328.419,Z 1174.299,A -85,B 0,C 180,E1 14839.122,E2 14839.122} C_VEL
LIN {X 0,Y 329.102,Z 1170.631,A -85,B 0,C 180,E1 14835.576,E2 14835.576} C_VEL
LIN {X 0,Y 330.52,Z 1165.163,A -85,B 0,C 180,E1 14831.482,E2 14831.482} C_VEL
LIN {X 0,Y 333.047,Z 1157.469,A -85,B 0,C 180,E1 14827.03,E2 14827.03} C_VEL
LIN {X 0,Y 336.102,Z 1149.666,A -85,B 0,C 180,E1 14823.309,E2 14823.309} C_VEL
LIN {X 0,Y 340.744,Z 1139.217,A -85,B 0,C 180,E1 14819.104,E2 14819.104} C_VEL
LIN {X 0,Y 346.414,Z 1127.298,A -85,B 0,C 180,E1 14815.148,E2 14815.148} C_VEL
LIN {X 0,Y 351.757,Z 1116.658,A -85,B 0,C 180,E1 14812.088,E2 14812.088} C_VEL
LIN {X 0,Y 352.896,Z 1113.002,A -85,B 0,C 180,E1 14810.99,E2 14810.99} C_VEL
LIN {X 0,Y 353.138,Z 1103.459,A -85,B 0,C 180,E1 14807.913,E2 14807.913} C_VEL
LIN {X 0,Y 354.458,Z 1099.893,A -85,B 0,C 180,E1 14807.023,E2 14807.023} C_VEL
LIN {X 0,Y 363.148,Z 1084.01,A -85,B 0,C 180,E1 14803.718,E2 14803.718} C_VEL
LIN {X 0,Y 372.621,Z 1066.047,A -85,B 0,C 180,E1 14800.593,E2 14800.593} C_VEL
LIN {X 0,Y 382.266,Z 1047.412,A -85,B 0,C 180,E1 14797.824,E2 14797.824} C_VEL
LIN {X 0,Y 391.523,Z 1028.471,A -85,B 0,C 180,E1 14795.449,E2 14795.449} C_VEL
LIN {X 0,Y 401.66,Z 1006.521,A -85,B 0,C 180,E1 14793.109,E2 14793.109} C_VEL
LIN {X 0,Y 409.845,Z 987.303,A -85,B 0,C 180,E1 14791.368,E2 14791.368} C_VEL
LIN {X 0,Y 418.971,Z 964.054,A -85,B 0,C 180,E1 14789.573,E2 14789.573} C_VEL
LIN {X 0,Y 426.506,Z 942.629,A -85,B 0,C 180,E1 14788.183,E2 14788.183} C_VEL
LIN {X 0,Y 434.293,Z 917.669,A -85,B 0,C 180,E1 14786.825,E2 14786.825} C_VEL
LIN {X 0,Y 440.359,Z 895.157,A -85,B 0,C 180,E1 14785.808,E2 14785.808} C_VEL
LIN {X 0,Y 446.296,Z 868.844,A -85,B 0,C 180,E1 14784.842,E2 14784.842} C_VEL
LIN {X 0,Y 453.894,Z 829.074,A -85,B 0,C 180,E1 14783.717,E2 14783.717} C_VEL
LIN {X 0,Y 467.074,Z 757.175,A -85,B 0,C 180,E1 14782.053,E2 14782.053} C_VEL
LIN {X 0,Y 478.043,Z 690.275,A -85,B 0,C 180,E1 14780.679,E2 14780.679} C_VEL
LIN {X 0,Y 487.18,Z 625.609,A -85,B 0,C 180,E1 14779.487,E2 14779.487} C_VEL
LIN {X 0,Y 492.708,Z 578.473,A -85,B 0,C 180,E1 14778.671,E2 14778.671} C_VEL
LIN {X 0,Y 489.074,Z 575.574,A -85,B 0,C 180,E1 14777.122,E2 14777.122} C_VEL
LIN {X 0,Y 482.097,Z 572.328,A -85,B 0,C 180,E1 14773.799,E2 14773.799} C_VEL
LIN {X 0,Y 475.775,Z 570.578,A -85,B 0,C 180,E1 14769.923,E2 14769.923} C_VEL
LIN {X 0,Y 471.023,Z 572.585,A -85,B 0,C 180,E1 14765.848,E2 14765.848} C_VEL
LIN {X 0,Y 468.952,Z 575.708,A -85,B 0,C 180,E1 14763.056,E2 14763.056} C_VEL
LIN {X 0,Y 467.746,Z 580.96,A -85,B 0,C 180,E1 14759.816,E2 14759.816} C_VEL
LIN {X 0,Y 467.933,Z 590.008,A -85,B 0,C 180,E1 14755.933,E2 14755.933} C_VEL
LIN {X 0,Y 465.936,Z 621.892,A -85,B 0,C 180,E1 14753.488,E2 14753.488} C_VEL
LIN {X 0,Y 464.393,Z 655.964,A -85,B 0,C 180,E1 14751.058,E2 14751.058} C_VEL
LIN {X 0,Y 463.138,Z 690.043,A -85,B 0,C 180,E1 14748.644,E2 14748.644} C_VEL
LIN {X 0,Y 462.897,Z 714.775,A -85,B 0,C 180,E1 14746.636,E2 14746.636} C_VEL
LIN {X 0,Y 463.51,Z 739.436,A -85,B 0,C 180,E1 14744.388,E2 14744.388} C_VEL
LIN {X 0,Y 465.199,Z 761.687,A -85,B 0,C 180,E1 14742.083,E2 14742.083} C_VEL
LIN {X 0,Y 467.862,Z 781.392,A -85,B 0,C 180,E1 14739.825,E2 14739.825} C_VEL
LIN {X 0,Y 470.57,Z 795.928,A -85,B 0,C 180,E1 14738.052,E2 14738.052} C_VEL
LIN {X 0,Y 462.74,Z 835.938,A -85,B 0,C 180,E1 14737.153,E2 14737.153} C_VEL
LIN {X 0,Y 453.999,Z 873.809,A -85,B 0,C 180,E1 14736.146,E2 14736.146} C_VEL
LIN {X 0,Y 445.264,Z 908.461,A -85,B 0,C 180,E1 14734.967,E2 14734.967} C_VEL
LIN {X 0,Y 436.12,Z 941.988,A -85,B 0,C 180,E1 14733.541,E2 14733.541} C_VEL
LIN {X 0,Y 427.011,Z 973.388,A -85,B 0,C 180,E1 14731.923,E2 14731.923} C_VEL
LIN {X 0,Y 419.727,Z 995.749,A -85,B 0,C 180,E1 14730.536,E2 14730.536} C_VEL
LIN {X 0,Y 411.901,Z 1016.862,A -85,B 0,C 180,E1 14728.966,E2 14728.966} C_VEL
LIN {X 0,Y 403.762,Z 1036.885,A -85,B 0,C 180,E1 14727.22,E2 14727.22} C_VEL
LIN {X 0,Y 394.762,Z 1056.846,A -85,B 0,C 180,E1 14725.146,E2 14725.146} C_VEL
LIN {X 0,Y 385.946,Z 1074.823,A -85,B 0,C 180,E1 14722.931,E2 14722.931} C_VEL
LIN {X 0,Y 377.059,Z 1091.952,A -85,B 0,C 180,E1 14720.473,E2 14720.473} C_VEL
LIN {X 0,Y 367.711,Z 1108.777,A -85,B 0,C 180,E1 14717.595,E2 14717.595} C_VEL
LIN {X 0,Y 358.853,Z 1123.974,A -85,B 0,C 180,E1 14714.495,E2 14714.495} C_VEL
LIN {X 0,Y 350.333,Z 1138.289,A -85,B 0,C 180,E1 14711.026,E2 14711.026} C_VEL
LIN {X 0,Y 342.751,Z 1150.925,A -85,B 0,C 180,E1 14707.354,E2 14707.354} C_VEL
LIN {X 0,Y 335.511,Z 1163.086,A -85,B 0,C 180,E1 14703.047,E2 14703.047} C_VEL
LIN {X 0,Y 329.801,Z 1173.201,A -85,B 0,C 180,E1 14698.619,E2 14698.619} C_VEL
LIN {X 0,Y 325.56,Z 1181.51,A -85,B 0,C 180,E1 14694.107,E2 14694.107} C_VEL
LIN {X 0,Y 322.578,Z 1188.409,A -85,B 0,C 180,E1 14689.367,E2 14689.367} C_VEL
LIN {X 0,Y 320.885,Z 1193.669,A -85,B 0,C 180,E1 14684.617,E2 14684.617} C_VEL
LIN {X 0,Y 320.156,Z 1197.292,A -85,B 0,C 180,E1 14680.07,E2 14680.07} C_VEL
LIN {X 0,Y 319.98,Z 1199.373,A -85,B 0,C 180,E1 14675.917,E2 14675.917} C_VEL
LIN {X 0,Y 319.977,Z 1200.376,A -85,B 0,C 180,E1 14671.788,E2 14671.788} C_VEL
LIN {X 0,Y 319.973,Z 1200.345,A -85,B 0,C 180,E1 14667.849,E2 14667.849} C_VEL
LIN {X 0,Y 319.984,Z 1199.225,A -85,B 0,C 180,E1 14663.719,E2 14663.719} C_VEL
LIN {X 0,Y 320.204,Z 1196.924,A -85,B 0,C 180,E1 14659.381,E2 14659.381} C_VEL
LIN {X 0,Y 321.027,Z 1193.161,A -85,B 0,C 180,E1 14654.831,E2 14654.831} C_VEL
LIN {X 0,Y 322.853,Z 1187.703,A -85,B 0,C 180,E1 14650.08,E2 14650.08} C_VEL
LIN {X 0,Y 325.989,Z 1180.585,A -85,B 0,C 180,E1 14645.343,E2 14645.343} C_VEL
LIN {X 0,Y 330.77,Z 1171.377,A -85,B 0,C 180,E1 14640.529,E2 14640.529} C_VEL
LIN {X 0,Y 336.83,Z 1160.737,A -85,B 0,C 180,E1 14636.075,E2 14636.075} C_VEL
LIN {X 0,Y 344.036,Z 1148.698,A -85,B 0,C 180,E1 14631.963,E2 14631.963} C_VEL
LIN {X 0,Y 352.222,Z 1135.133,A -85,B 0,C 180,E1 14628.153,E2 14628.153} C_VEL
LIN {X 0,Y 361.208,Z 1120.039,A -85,B 0,C 180,E1 14624.647,E2 14624.647} C_VEL
LIN {X 0,Y 370.274,Z 1104.165,A -85,B 0,C 180,E1 14621.58,E2 14621.58} C_VEL
LIN {X 0,Y 380.023,Z 1086.239,A -85,B 0,C 180,E1 14618.67,E2 14618.67} C_VEL
LIN {X 0,Y 390.012,Z 1066.606,A -85,B 0,C 180,E1 14616.013,E2 14616.013} C_VEL
LIN {X 0,Y 399.624,Z 1046.098,A -85,B 0,C 180,E1 14613.7,E2 14613.7} C_VEL
LIN {X 0,Y 408.85,Z 1024.517,A -85,B 0,C 180,E1 14611.67,E2 14611.67} C_VEL
LIN {X 0,Y 417.205,Z 1002.645,A -85,B 0,C 180,E1 14609.957,E2 14609.957} C_VEL
LIN {X 0,Y 425.189,Z 978.953,A -85,B 0,C 180,E1 14608.415,E2 14608.415} C_VEL
LIN {X 0,Y 434.423,Z 947.714,A -85,B 0,C 180,E1 14606.74,E2 14606.74} C_VEL
LIN {X 0,Y 444.003,Z 912.843,A -85,B 0,C 180,E1 14605.21,E2 14605.21} C_VEL
LIN {X 0,Y 452.837,Z 878.134,A -85,B 0,C 180,E1 14603.993,E2 14603.993} C_VEL
LIN {X 0,Y 461.785,Z 839.899,A -85,B 0,C 180,E1 14602.949,E2 14602.949} C_VEL
LIN {X 0,Y 470.422,Z 796.198,A -85,B 0,C 180,E1 14601.96,E2 14601.96} C_VEL
LIN {X 0,Y 477.158,Z 754.163,A -85,B 0,C 180,E1 14601.164,E2 14601.164} C_VEL
LIN {X 0,Y 480.429,Z 729.281,A -85,B 0,C 180,E1 14600.742,E2 14600.742} C_VEL
LIN {X 0,Y 473.606,Z 748.245,A -85,B 0,C 180,E1 14599.767,E2 14599.767} C_VEL
LIN {X 0,Y 470.779,Z 755.727,A -85,B 0,C 180,E1 14599.358,E2 14599.358} C_VEL
LIN {X 0,Y 463.402,Z 775.552,A -85,B 0,C 180,E1 14598.411,E2 14598.411} C_VEL
LIN {X 0,Y 457.349,Z 790.013,A -85,B 0,C 180,E1 14597.56,E2 14597.56} C_VEL
LIN {X 0,Y 449.996,Z 807.983,A -85,B 0,C 180,E1 14596.624,E2 14596.624} C_VEL
LIN {X 0,Y 444.898,Z 819.34,A -85,B 0,C 180,E1 14595.905,E2 14595.905} C_VEL
LIN {X 0,Y 437.522,Z 836.215,A -85,B 0,C 180,E1 14594.958,E2 14594.958} C_VEL
LIN {X 0,Y 433.053,Z 845.794,A -85,B 0,C 180,E1 14594.314,E2 14594.314} C_VEL
LIN {X 0,Y 425.917,Z 861.431,A -85,B 0,C 180,E1 14593.37,E2 14593.37} C_VEL
LIN {X 0,Y 421.624,Z 870.317,A -85,B 0,C 180,E1 14592.742,E2 14592.742} C_VEL
LIN {X 0,Y 414.701,Z 885.098,A -85,B 0,C 180,E1 14591.784,E2 14591.784} C_VEL
LIN {X 0,Y 411.838,Z 890.964,A -85,B 0,C 180,E1 14591.342,E2 14591.342} C_VEL
LIN {X 0,Y 404.481,Z 906.864,A -85,B 0,C 180,E1 14590.397,E2 14590.397} C_VEL
LIN {X 0,Y 402.672,Z 910.726,A -85,B 0,C 180,E1 14590.155,E2 14590.155} C_VEL
LIN {X 0,Y 396.805,Z 924.131,A -85,B 0,C 180,E1 14589.573,E2 14589.573} C_VEL
LIN {X 0,Y 393.803,Z 930.54,A -85,B 0,C 180,E1 14589.234,E2 14589.234} C_VEL
LIN {X 0,Y 387.931,Z 943.116,A -85,B 0,C 180,E1 14588.672,E2 14588.672} C_VEL
LIN {X 0,Y 383.9,Z 950.83,A -85,B 0,C 180,E1 14588.211,E2 14588.211} C_VEL
LIN {X 0,Y 378.35,Z 961.132,A -85,B 0,C 180,E1 14587.67,E2 14587.67} C_VEL
LIN {X 0,Y 374.972,Z 966.987,A -85,B 0,C 180,E1 14587.26,E2 14587.26} C_VEL
LIN {X 0,Y 369.399,Z 976.23,A -85,B 0,C 180,E1 14586.684,E2 14586.684} C_VEL
LIN {X 0,Y 366.116,Z 981.464,A -85,B 0,C 180,E1 14586.272,E2 14586.272} C_VEL
LIN {X 0,Y 360.711,Z 989.584,A -85,B 0,C 180,E1 14585.637,E2 14585.637} C_VEL
LIN {X 0,Y 358.521,Z 992.795,A -85,B 0,C 180,E1 14585.336,E2 14585.336} C_VEL
LIN {X 0,Y 354.216,Z 998.895,A -85,B 0,C 180,E1 14584.811,E2 14584.811} C_VEL
LIN {X 0,Y 351.49,Z 1002.605,A -85,B 0,C 180,E1 14584.405,E2 14584.405} C_VEL
LIN {X 0,Y 347.153,Z 1008.416,A -85,B 0,C 180,E1 14583.798,E2 14583.798} C_VEL
LIN {X 0,Y 345.212,Z 1010.917,A -85,B 0,C 180,E1 14583.487,E2 14583.487} C_VEL
LIN {X 0,Y 341.404,Z 1015.758,A -85,B 0,C 180,E1 14582.891,E2 14582.891} C_VEL
LIN {X 0,Y 339.811,Z 1017.665,A -85,B 0,C 180,E1 14582.57,E2 14582.57} C_VEL
LIN {X 0,Y 337.212,Z 1020.916,A -85,B 0,C 180,E1 14582.172,E2 14582.172} C_VEL
LIN {X 0,Y 335.117,Z 1023.569,A -85,B 0,C 180,E1 14581.601,E2 14581.601} C_VEL
LIN {X 0,Y 334.429,Z 1037.485,A -85,B 0,C 180,E1 14580.685,E2 14580.685} C_VEL
LIN {X 0,Y 333.385,Z 1050.825,A -85,B 0,C 180,E1 14579.484,E2 14579.484} C_VEL
LIN {X 0,Y 332.309,Z 1061.325,A -85,B 0,C 180,E1 14578.276,E2 14578.276} C_VEL
LIN {X 0,Y 330.951,Z 1072.281,A -85,B 0,C 180,E1 14576.709,E2 14576.709} C_VEL
LIN {X 0,Y 329.495,Z 1081.764,A -85,B 0,C 180,E1 14574.951,E2 14574.951} C_VEL
LIN {X 0,Y 328.234,Z 1088.919,A -85,B 0,C 180,E1 14573.269,E2 14573.269} C_VEL
LIN {X 0,Y 327.106,Z 1094.709,A -85,B 0,C 180,E1 14571.563,E2 14571.563} C_VEL
LIN {X 0,Y 326.076,Z 1099.43,A -85,B 0,C 180,E1 14569.755,E2 14569.755} C_VEL
LIN {X 0,Y 325.074,Z 1103.52,A -85,B 0,C 180,E1 14567.566,E2 14567.566} C_VEL
LIN {X 0,Y 324.234,Z 1105.99,A -85,B 0,C 180,E1 14565.169,E2 14565.169} C_VEL
LIN {X 0,Y 323.751,Z 1106.676,A -85,B 0,C 180,E1 14563.123,E2 14563.123} C_VEL
LIN {X 0,Y 323.48,Z 1106.207,A -85,B 0,C 180,E1 14561.248,E2 14561.248} C_VEL
LIN {X 0,Y 323.376,Z 1104.652,A -85,B 0,C 180,E1 14559.36,E2 14559.36} C_VEL
LIN {X 0,Y 323.424,Z 1101.974,A -85,B 0,C 180,E1 14557.458,E2 14557.458} C_VEL
LIN {X 0,Y 323.687,Z 1097.658,A -85,B 0,C 180,E1 14555.353,E2 14555.353} C_VEL
LIN {X 0,Y 324.209,Z 1091.103,A -85,B 0,C 180,E1 14553.04,E2 14553.04} C_VEL
LIN {X 0,Y 324.847,Z 1083.796,A -85,B 0,C 180,E1 14551.102,E2 14551.102} C_VEL
LIN {X 0,Y 325.609,Z 1075.366,A -85,B 0,C 180,E1 14549.301,E2 14549.301} C_VEL
LIN {X 0,Y 325.84,Z 1073.209,A -85,B 0,C 180,E1 14548.86,E2 14548.86} C_VEL
LIN {X 0,Y 327.484,Z 1073.697,A -85,B 0,C 180,E1 14548.115,E2 14548.115} C_VEL
LIN {X 0,Y 329.069,Z 1073.603,A -85,B 0,C 180,E1 14547.644,E2 14547.644} C_VEL
LIN {X 0,Y 335.559,Z 1073.531,A -85,B 0,C 180,E1 14545.724,E2 14545.724} C_VEL
LIN {X 0,Y 343.484,Z 1072.981,A -85,B 0,C 180,E1 14543.776,E2 14543.776} C_VEL
LIN {X 0,Y 355.766,Z 1071.205,A -85,B 0,C 180,E1 14541.395,E2 14541.395} C_VEL
LIN {X 0,Y 369.546,Z 1068.324,A -85,B 0,C 180,E1 14539.301,E2 14539.301} C_VEL
LIN {X 0,Y 371.627,Z 1067.838,A -85,B 0,C 180,E1 14539.017,E2 14539.017} C_VEL
LIN {X 0,Y 361.778,Z 1086.373,A -85,B 0,C 180,E1 14535.713,E2 14535.713} C_VEL
LIN {X 0,Y 353.585,Z 1101.475,A -85,B 0,C 180,E1 14532.523,E2 14532.523} C_VEL
LIN {X 0,Y 344.639,Z 1117.998,A -85,B 0,C 180,E1 14528.382,E2 14528.382} C_VEL
LIN {X 0,Y 338.053,Z 1130.618,A -85,B 0,C 180,E1 14524.606,E2 14524.606} C_VEL
LIN {X 0,Y 331.888,Z 1143.014,A -85,B 0,C 180,E1 14520.156,E2 14520.156} C_VEL
LIN {X 0,Y 327.758,Z 1152.135,A -85,B 0,C 180,E1 14516.245,E2 14516.245} C_VEL
LIN {X 0,Y 324.172,Z 1161.165,A -85,B 0,C 180,E1 14511.536,E2 14511.536} C_VEL
LIN {X 0,Y 322.217,Z 1167.078,A -85,B 0,C 180,E1 14507.698,E2 14507.698} C_VEL
LIN {X 0,Y 320.991,Z 1171.815,A -85,B 0,C 180,E1 14503.88,E2 14503.88} C_VEL
LIN {X 0,Y 320.274,Z 1176.006,A -85,B 0,C 180,E1 14499.345,E2 14499.345} C_VEL
LIN {X 0,Y 320.035,Z 1178.258,A -85,B 0,C 180,E1 14495.38,E2 14495.38} C_VEL
LIN {X 0,Y 319.982,Z 1179.255,A -85,B 0,C 180,E1 14491.972,E2 14491.972} C_VEL
LIN {X 0,Y 319.98,Z 1179.36,A -85,B 0,C 180,E1 14488.749,E2 14488.749} C_VEL
LIN {X 0,Y 320.013,Z 1178.57,A -85,B 0,C 180,E1 14485.343,E2 14485.343} C_VEL
LIN {X 0,Y 320.159,Z 1176.854,A -85,B 0,C 180,E1 14481.903,E2 14481.903} C_VEL
LIN {X 0,Y 320.53,Z 1174.156,A -85,B 0,C 180,E1 14478.386,E2 14478.386} C_VEL
LIN {X 0,Y 321.474,Z 1169.874,A -85,B 0,C 180,E1 14474.303,E2 14474.303} C_VEL
LIN {X 0,Y 323.382,Z 1163.426,A -85,B 0,C 180,E1 14469.741,E2 14469.741} C_VEL
LIN {X 0,Y 325.877,Z 1156.7,A -85,B 0,C 180,E1 14465.918,E2 14465.918} C_VEL
LIN {X 0,Y 329.893,Z 1147.443,A -85,B 0,C 180,E1 14461.52,E2 14461.52} C_VEL
LIN {X 0,Y 335.086,Z 1136.475,A -85,B 0,C 180,E1 14457.298,E2 14457.298} C_VEL
LIN {X 0,Y 341.373,Z 1124.316,A -85,B 0,C 180,E1 14453.311,E2 14453.311} C_VEL
LIN {X 0,Y 348.95,Z 1110.043,A -85,B 0,C 180,E1 14449.428,E2 14449.428} C_VEL
LIN {X 0,Y 354.458,Z 1099.893,A -85,B 0,C 180,E1 14447.023,E2 14447.023} C_VEL
LIN {X 0,Y 355.98,Z 1095.859,A -85,B 0,C 180,E1 14445.989,E2 14445.989} C_VEL
LIN {X 0,Y 357.426,Z 1085.3,A -85,B 0,C 180,E1 14443.033,E2 14443.033} C_VEL
LIN {X 0,Y 359.048,Z 1081.388,A -85,B 0,C 180,E1 14442.209,E2 14442.209} C_VEL
LIN {X 0,Y 367.796,Z 1065.512,A -85,B 0,C 180,E1 14439.463,E2 14439.463} C_VEL
LIN {X 0,Y 378.367,Z 1045.622,A -85,B 0,C 180,E1 14436.552,E2 14436.552} C_VEL
LIN {X 0,Y 387.012,Z 1028.463,A -85,B 0,C 180,E1 14434.413,E2 14434.413} C_VEL
LIN {X 0,Y 397.244,Z 1006.872,A -85,B 0,C 180,E1 14432.119,E2 14432.119} C_VEL
LIN {X 0,Y 405.661,Z 987.727,A -85,B 0,C 180,E1 14430.385,E2 14430.385} C_VEL
LIN {X 0,Y 415.051,Z 964.3,A -85,B 0,C 180,E1 14428.59,E2 14428.59} C_VEL
LIN {X 0,Y 422.74,Z 943.009,A -85,B 0,C 180,E1 14427.215,E2 14427.215} C_VEL
LIN {X 0,Y 430.56,Z 918.397,A -85,B 0,C 180,E1 14425.887,E2 14425.887} C_VEL
LIN {X 0,Y 436.731,Z 896.1,A -85,B 0,C 180,E1 14424.883,E2 14424.883} C_VEL
LIN {X 0,Y 442.676,Z 870.269,A -85,B 0,C 180,E1 14423.94,E2 14423.94} C_VEL
LIN {X 0,Y 450.58,Z 829.899,A -85,B 0,C 180,E1 14422.8,E2 14422.8} C_VEL
LIN {X 0,Y 463.584,Z 761.053,A -85,B 0,C 180,E1 14421.209,E2 14421.209} C_VEL
LIN {X 0,Y 474.91,Z 693.831,A -85,B 0,C 180,E1 14419.832,E2 14419.832} C_VEL
LIN {X 0,Y 484.304,Z 628.796,A -85,B 0,C 180,E1 14418.64,E2 14418.64} C_VEL
LIN {X 0,Y 489.605,Z 584.985,A -85,B 0,C 180,E1 14417.891,E2 14417.891} C_VEL
LIN {X 0,Y 487.181,Z 583.172,A -85,B 0,C 180,E1 14416.821,E2 14416.821} C_VEL
LIN {X 0,Y 480.806,Z 580.208,A -85,B 0,C 180,E1 14413.714,E2 14413.714} C_VEL
LIN {X 0,Y 474.764,Z 578.52,A -85,B 0,C 180,E1 14409.945,E2 14409.945} C_VEL
LIN {X 0,Y 470.037,Z 580.619,A -85,B 0,C 180,E1 14405.861,E2 14405.861} C_VEL
LIN {X 0,Y 468.034,Z 583.599,A -85,B 0,C 180,E1 14403.184,E2 14403.184} C_VEL
LIN {X 0,Y 466.779,Z 588.774,A -85,B 0,C 180,E1 14400,E2 14400} C_VEL
LIN {X 0,Y 466.752,Z 596.794,A -85,B 0,C 180,E1 14396.546,E2 14396.546} C_VEL
LIN {X 0,Y 464.395,Z 630.791,A -85,B 0,C 180,E1 14393.964,E2 14393.964} C_VEL
LIN {X 0,Y 462.347,Z 667.208,A -85,B 0,C 180,E1 14391.387,E2 14391.387} C_VEL
LIN {X 0,Y 461.015,Z 696.304,A -85,B 0,C 180,E1 14389.293,E2 14389.293} C_VEL
LIN {X 0,Y 460.475,Z 723.104,A -85,B 0,C 180,E1 14387.076,E2 14387.076} C_VEL
LIN {X 0,Y 460.925,Z 747.596,A -85,B 0,C 180,E1 14384.766,E2 14384.766} C_VEL
LIN {X 0,Y 462.29,Z 767.931,A -85,B 0,C 180,E1 14382.617,E2 14382.617} C_VEL
LIN {X 0,Y 464.575,Z 787.009,A -85,B 0,C 180,E1 14380.398,E2 14380.398} C_VEL
LIN {X 0,Y 466.668,Z 799.42,A -85,B 0,C 180,E1 14378.874,E2 14378.874} C_VEL
LIN {X 0,Y 457.687,Z 843.195,A -85,B 0,C 180,E1 14377.879,E2 14377.879} C_VEL
LIN {X 0,Y 448.98,Z 879.406,A -85,B 0,C 180,E1 14376.885,E2 14376.885} C_VEL
LIN {X 0,Y 439.628,Z 915.213,A -85,B 0,C 180,E1 14375.624,E2 14375.624} C_VEL
LIN {X 0,Y 430.396,Z 948.05,A -85,B 0,C 180,E1 14374.183,E2 14374.183} C_VEL
LIN {X 0,Y 421.928,Z 976.099,A -85,B 0,C 180,E1 14372.702,E2 14372.702} C_VEL
LIN {X 0,Y 414.694,Z 997.566,A -85,B 0,C 180,E1 14371.356,E2 14371.356} C_VEL
LIN {X 0,Y 406.056,Z 1020.015,A -85,B 0,C 180,E1 14369.66,E2 14369.66} C_VEL
LIN {X 0,Y 397.317,Z 1040.218,A -85,B 0,C 180,E1 14367.828,E2 14367.828} C_VEL
LIN {X 0,Y 388.233,Z 1059.596,A -85,B 0,C 180,E1 14365.76,E2 14365.76} C_VEL
LIN {X 0,Y 378.566,Z 1078.604,A -85,B 0,C 180,E1 14363.35,E2 14363.35} C_VEL
LIN {X 0,Y 368.912,Z 1096.099,A -85,B 0,C 180,E1 14360.693,E2 14360.693} C_VEL
LIN {X 0,Y 358.916,Z 1113.335,A -85,B 0,C 180,E1 14357.579,E2 14357.579} C_VEL
LIN {X 0,Y 349.618,Z 1128.656,A -85,B 0,C 180,E1 14354.249,E2 14354.249} C_VEL
LIN {X 0,Y 340.854,Z 1142.806,A -85,B 0,C 180,E1 14350.555,E2 14350.555} C_VEL
LIN {X 0,Y 332.828,Z 1155.543,A -85,B 0,C 180,E1 14346.498,E2 14346.498} C_VEL
LIN {X 0,Y 326.387,Z 1166.037,A -85,B 0,C 180,E1 14342.416,E2 14342.416} C_VEL
LIN {X 0,Y 320.677,Z 1175.982,A -85,B 0,C 180,E1 14337.683,E2 14337.683} C_VEL
LIN {X 0,Y 316.455,Z 1184.289,A -85,B 0,C 180,E1 14332.671,E2 14332.671} C_VEL
LIN {X 0,Y 313.829,Z 1190.632,A -85,B 0,C 180,E1 14327.702,E2 14327.702} C_VEL
LIN {X 0,Y 312.547,Z 1195.016,A -85,B 0,C 180,E1 14323.126,E2 14323.126} C_VEL
LIN {X 0,Y 312.062,Z 1197.952,A -85,B 0,C 180,E1 14318.659,E2 14318.659} C_VEL
LIN {X 0,Y 311.97,Z 1199.625,A -85,B 0,C 180,E1 14314.409,E2 14314.409} C_VEL
LIN {X 0,Y 311.976,Z 1200.228,A -85,B 0,C 180,E1 14310.365,E2 14310.365} C_VEL
LIN {X 0,Y 311.973,Z 1199.801,A -85,B 0,C 180,E1 14306.323,E2 14306.323} C_VEL
LIN {X 0,Y 312.03,Z 1198.355,A -85,B 0,C 180,E1 14302.078,E2 14302.078} C_VEL
LIN {X 0,Y 312.422,Z 1195.557,A -85,B 0,C 180,E1 14297.616,E2 14297.616} C_VEL
LIN {X 0,Y 313.666,Z 1191.113,A -85,B 0,C 180,E1 14292.753,E2 14292.753} C_VEL
LIN {X 0,Y 316.212,Z 1184.816,A -85,B 0,C 180,E1 14287.698,E2 14287.698} C_VEL
LIN {X 0,Y 320.129,Z 1176.999,A -85,B 0,C 180,E1 14282.868,E2 14282.868} C_VEL
LIN {X 0,Y 325.398,Z 1167.717,A -85,B 0,C 180,E1 14278.299,E2 14278.299} C_VEL
LIN {X 0,Y 332.224,Z 1156.514,A -85,B 0,C 180,E1 14273.848,E2 14273.848} C_VEL
LIN {X 0,Y 340.245,Z 1143.698,A -85,B 0,C 180,E1 14269.718,E2 14269.718} C_VEL
LIN {X 0,Y 349.209,Z 1129.287,A -85,B 0,C 180,E1 14265.909,E2 14265.909} C_VEL
LIN {X 0,Y 358.456,Z 1114.045,A -85,B 0,C 180,E1 14262.571,E2 14262.571} C_VEL
LIN {X 0,Y 368.663,Z 1096.512,A -85,B 0,C 180,E1 14259.376,E2 14259.376} C_VEL
LIN {X 0,Y 378.692,Z 1078.25,A -85,B 0,C 180,E1 14256.612,E2 14256.612} C_VEL
LIN {X 0,Y 388.823,Z 1058.314,A -85,B 0,C 180,E1 14254.098,E2 14254.098} C_VEL
LIN {X 0,Y 398.319,Z 1037.912,A -85,B 0,C 180,E1 14251.952,E2 14251.952} C_VEL
LIN {X 0,Y 407.637,Z 1015.829,A -85,B 0,C 180,E1 14250.016,E2 14250.016} C_VEL
LIN {X 0,Y 416,Z 993.666,A -85,B 0,C 180,E1 14248.391,E2 14248.391} C_VEL
LIN {X 0,Y 423.937,Z 969.579,A -85,B 0,C 180,E1 14246.93,E2 14246.93} C_VEL
LIN {X 0,Y 433.741,Z 935.974,A -85,B 0,C 180,E1 14245.264,E2 14245.264} C_VEL
LIN {X 0,Y 442.557,Z 903.94,A -85,B 0,C 180,E1 14243.955,E2 14243.955} C_VEL
LIN {X 0,Y 451.505,Z 868.817,A -85,B 0,C 180,E1 14242.802,E2 14242.802} C_VEL
LIN {X 0,Y 460.732,Z 828.786,A -85,B 0,C 180,E1 14241.786,E2 14241.786} C_VEL
LIN {X 0,Y 468.914,Z 786.205,A -85,B 0,C 180,E1 14240.859,E2 14240.859} C_VEL
LIN {X 0,Y 473.682,Z 756.704,A -85,B 0,C 180,E1 14240.306,E2 14240.306} C_VEL
LIN {X 0,Y 465.694,Z 778.009,A -85,B 0,C 180,E1 14239.325,E2 14239.325} C_VEL
LIN {X 0,Y 458.94,Z 793.909,A -85,B 0,C 180,E1 14238.416,E2 14238.416} C_VEL
LIN {X 0,Y 451.282,Z 812.12,A -85,B 0,C 180,E1 14237.479,E2 14237.479} C_VEL
LIN {X 0,Y 446.16,Z 823.311,A -85,B 0,C 180,E1 14236.789,E2 14236.789} C_VEL
LIN {X 0,Y 438.494,Z 840.401,A -85,B 0,C 180,E1 14235.841,E2 14235.841} C_VEL
LIN {X 0,Y 433.984,Z 849.785,A -85,B 0,C 180,E1 14235.228,E2 14235.228} C_VEL
LIN {X 0,Y 426.773,Z 865.218,A -85,B 0,C 180,E1 14234.311,E2 14234.311} C_VEL
LIN {X 0,Y 422.371,Z 874.133,A -85,B 0,C 180,E1 14233.694,E2 14233.694} C_VEL
LIN {X 0,Y 415.197,Z 888.963,A -85,B 0,C 180,E1 14232.749,E2 14232.749} C_VEL
LIN {X 0,Y 412.296,Z 894.833,A -85,B 0,C 180,E1 14232.323,E2 14232.323} C_VEL
LIN {X 0,Y 404.339,Z 911.457,A -85,B 0,C 180,E1 14231.338,E2 14231.338} C_VEL
LIN {X 0,Y 401.706,Z 917.389,A -85,B 0,C 180,E1 14231.084,E2 14231.084} C_VEL
LIN {X 0,Y 395.511,Z 930.647,A -85,B 0,C 180,E1 14230.44,E2 14230.44} C_VEL
LIN {X 0,Y 388.301,Z 945.79,A -85,B 0,C 180,E1 14229.785,E2 14229.785} C_VEL
LIN {X 0,Y 384.039,Z 953.824,A -85,B 0,C 180,E1 14229.324,E2 14229.324} C_VEL
LIN {X 0,Y 377.924,Z 964.772,A -85,B 0,C 180,E1 14228.751,E2 14228.751} C_VEL
LIN {X 0,Y 374.453,Z 970.62,A -85,B 0,C 180,E1 14228.369,E2 14228.369} C_VEL
LIN {X 0,Y 368.323,Z 980.421,A -85,B 0,C 180,E1 14227.741,E2 14227.741} C_VEL
LIN {X 0,Y 364.986,Z 985.437,A -85,B 0,C 180,E1 14227.375,E2 14227.375} C_VEL
LIN {X 0,Y 359.354,Z 993.676,A -85,B 0,C 180,E1 14226.711,E2 14226.711} C_VEL
LIN {X 0,Y 352.358,Z 1003.257,A -85,B 0,C 180,E1 14225.863,E2 14225.863} C_VEL
LIN {X 0,Y 345.732,Z 1011.866,A -85,B 0,C 180,E1 14224.977,E2 14224.977} C_VEL
LIN {X 0,Y 343.068,Z 1015.194,A -85,B 0,C 180,E1 14224.588,E2 14224.588} C_VEL
LIN {X 0,Y 338.742,Z 1020.429,A -85,B 0,C 180,E1 14223.893,E2 14223.893} C_VEL
LIN {X 0,Y 333.965,Z 1026.052,A -85,B 0,C 180,E1 14223.089,E2 14223.089} C_VEL
LIN {X 0,Y 332.344,Z 1027.863,A -85,B 0,C 180,E1 14222.719,E2 14222.719} C_VEL
LIN {X 0,Y 329.205,Z 1031.496,A -85,B 0,C 180,E1 14222.161,E2 14222.161} C_VEL
LIN {X 0,Y 327.716,Z 1033.218,A -85,B 0,C 180,E1 14221.705,E2 14221.705} C_VEL
LIN {X 0,Y 326.89,Z 1044.688,A -85,B 0,C 180,E1 14220.789,E2 14220.789} C_VEL
LIN {X 0,Y 325.846,Z 1055.944,A -85,B 0,C 180,E1 14219.648,E2 14219.648} C_VEL
LIN {X 0,Y 324.277,Z 1068.79,A -85,B 0,C 180,E1 14217.968,E2 14217.968} C_VEL
LIN {X 0,Y 322.917,Z 1077.862,A -85,B 0,C 180,E1 14216.449,E2 14216.449} C_VEL
LIN {X 0,Y 321.571,Z 1085.692,A -85,B 0,C 180,E1 14214.826,E2 14214.826} C_VEL
LIN {X 0,Y 320.099,Z 1093.37,A -85,B 0,C 180,E1 14212.822,E2 14212.822} C_VEL
LIN {X 0,Y 318.668,Z 1099.497,A -85,B 0,C 180,E1 14210.61,E2 14210.61} C_VEL
LIN {X 0,Y 317.688,Z 1103.273,A -85,B 0,C 180,E1 14208.747,E2 14208.747} C_VEL
LIN {X 0,Y 316.892,Z 1105.888,A -85,B 0,C 180,E1 14206.869,E2 14206.869} C_VEL
LIN {X 0,Y 316.265,Z 1107.402,A -85,B 0,C 180,E1 14204.974,E2 14204.974} C_VEL
LIN {X 0,Y 315.806,Z 1107.839,A -85,B 0,C 180,E1 14202.98,E2 14202.98} C_VEL
LIN {X 0,Y 315.512,Z 1107.018,A -85,B 0,C 180,E1 14200.807,E2 14200.807} C_VEL
LIN {X 0,Y 315.455,Z 1104.306,A -85,B 0,C 180,E1 14198.232,E2 14198.232} C_VEL
LIN {X 0,Y 315.626,Z 1100.398,A -85,B 0,C 180,E1 14196.077,E2 14196.077} C_VEL
LIN {X 0,Y 315.975,Z 1095.517,A -85,B 0,C 180,E1 14194.107,E2 14194.107} C_VEL
LIN {X 0,Y 316.52,Z 1089.188,A -85,B 0,C 180,E1 14192.126,E2 14192.126} C_VEL
LIN {X 0,Y 317.354,Z 1080.281,A -85,B 0,C 180,E1 14189.936,E2 14189.936} C_VEL
LIN {X 0,Y 317.571,Z 1078.351,A -85,B 0,C 180,E1 14189.489,E2 14189.489} C_VEL
LIN {X 0,Y 319.301,Z 1078.829,A -85,B 0,C 180,E1 14188.679,E2 14188.679} C_VEL
LIN {X 0,Y 320.68,Z 1078.876,A -85,B 0,C 180,E1 14188.2,E2 14188.2} C_VEL
LIN {X 0,Y 329.519,Z 1079.035,A -85,B 0,C 180,E1 14185.428,E2 14185.428} C_VEL
LIN {X 0,Y 339.983,Z 1078.215,A -85,B 0,C 180,E1 14182.921,E2 14182.921} C_VEL
LIN {X 0,Y 351.812,Z 1076.536,A -85,B 0,C 180,E1 14180.669,E2 14180.669} C_VEL
LIN {X 0,Y 362.9,Z 1074.46,A -85,B 0,C 180,E1 14178.947,E2 14178.947} C_VEL
LIN {X 0,Y 353.798,Z 1090.628,A -85,B 0,C 180,E1 14175.879,E2 14175.879} C_VEL
LIN {X 0,Y 344.716,Z 1106.751,A -85,B 0,C 180,E1 14172.297,E2 14172.297} C_VEL
LIN {X 0,Y 336.799,Z 1120.73,A -85,B 0,C 180,E1 14168.57,E2 14168.57} C_VEL
LIN {X 0,Y 329.527,Z 1134.084,A -85,B 0,C 180,E1 14164.361,E2 14164.361} C_VEL
LIN {X 0,Y 323.892,Z 1144.979,A -85,B 0,C 180,E1 14160.214,E2 14160.214} C_VEL
LIN {X 0,Y 319.176,Z 1155.075,A -85,B 0,C 180,E1 14155.617,E2 14155.617} C_VEL
LIN {X 0,Y 316.053,Z 1162.645,A -85,B 0,C 180,E1 14151.337,E2 14151.337} C_VEL
LIN {X 0,Y 314.051,Z 1168.604,A -85,B 0,C 180,E1 14147.223,E2 14147.223} C_VEL
LIN {X 0,Y 312.686,Z 1173.95,A -85,B 0,C 180,E1 14142.374,E2 14142.374} C_VEL
LIN {X 0,Y 312.21,Z 1176.955,A -85,B 0,C 180,E1 14138.474,E2 14138.474} C_VEL
LIN {X 0,Y 312.027,Z 1178.728,A -85,B 0,C 180,E1 14134.966,E2 14134.966} C_VEL
LIN {X 0,Y 311.984,Z 1179.564,A -85,B 0,C 180,E1 14131.655,E2 14131.655} C_VEL
LIN {X 0,Y 311.984,Z 1179.577,A -85,B 0,C 180,E1 14128.349,E2 14128.349} C_VEL
LIN {X 0,Y 312.025,Z 1178.766,A -85,B 0,C 180,E1 14125.039,E2 14125.039} C_VEL
LIN {X 0,Y 312.202,Z 1177.019,A -85,B 0,C 180,E1 14121.531,E2 14121.531} C_VEL
LIN {X 0,Y 312.633,Z 1174.196,A -85,B 0,C 180,E1 14117.816,E2 14117.816} C_VEL
LIN {X 0,Y 313.875,Z 1169.245,A -85,B 0,C 180,E1 14113.151,E2 14113.151} C_VEL
LIN {X 0,Y 315.893,Z 1163.104,A -85,B 0,C 180,E1 14108.851,E2 14108.851} C_VEL
LIN {X 0,Y 318.634,Z 1156.295,A -85,B 0,C 180,E1 14104.938,E2 14104.938} C_VEL
LIN {X 0,Y 323.363,Z 1146.104,A -85,B 0,C 180,E1 14100.146,E2 14100.146} C_VEL
LIN {X 0,Y 328.329,Z 1136.316,A -85,B 0,C 180,E1 14096.343,E2 14096.343} C_VEL
LIN {X 0,Y 335.124,Z 1123.93,A -85,B 0,C 180,E1 14092.248,E2 14092.248} C_VEL
LIN {X 0,Y 342.647,Z 1110.36,A -85,B 0,C 180,E1 14088.519,E2 14088.519} C_VEL
LIN {X 0,Y 351.052,Z 1095.714,A -85,B 0,C 180,E1 14085.063,E2 14085.063} C_VEL
LIN {X 0,Y 359.048,Z 1081.388,A -85,B 0,C 180,E1 14082.209,E2 14082.209} C_VEL
LIN {X 0,Y 360.926,Z 1076.866,A -85,B 0,C 180,E1 14081.252,E2 14081.252} C_VEL
LIN {X 0,Y 363.471,Z 1065.351,A -85,B 0,C 180,E1 14078.457,E2 14078.457} C_VEL
LIN {X 0,Y 365.302,Z 1061.13,A -85,B 0,C 180,E1 14077.702,E2 14077.702} C_VEL
LIN {X 0,Y 374.368,Z 1044.38,A -85,B 0,C 180,E1 14075.323,E2 14075.323} C_VEL
LIN {X 0,Y 384.05,Z 1025.832,A -85,B 0,C 180,E1 14073.04,E2 14073.04} C_VEL
LIN {X 0,Y 393.898,Z 1005.252,A -85,B 0,C 180,E1 14070.913,E2 14070.913} C_VEL
LIN {X 0,Y 403.584,Z 983.636,A -85,B 0,C 180,E1 14069.011,E2 14069.011} C_VEL
LIN {X 0,Y 412.013,Z 962.637,A -85,B 0,C 180,E1 14067.458,E2 14067.458} C_VEL
LIN {X 0,Y 420.49,Z 939.418,A -85,B 0,C 180,E1 14065.998,E2 14065.998} C_VEL
LIN {X 0,Y 427.502,Z 917.309,A -85,B 0,C 180,E1 14064.844,E2 14064.844} C_VEL
LIN {X 0,Y 434.297,Z 892.837,A -85,B 0,C 180,E1 14063.776,E2 14063.776} C_VEL
LIN {X 0,Y 439.664,Z 869.309,A -85,B 0,C 180,E1 14062.946,E2 14062.946} C_VEL
LIN {X 0,Y 448.133,Z 827.34,A -85,B 0,C 180,E1 14061.781,E2 14061.781} C_VEL
LIN {X 0,Y 461.703,Z 756.747,A -85,B 0,C 180,E1 14060.176,E2 14060.176} C_VEL
LIN {X 0,Y 473.116,Z 689.571,A -85,B 0,C 180,E1 14058.826,E2 14058.826} C_VEL
LIN {X 0,Y 482.43,Z 625.168,A -85,B 0,C 180,E1 14057.666,E2 14057.666} C_VEL
LIN {X 0,Y 486.573,Z 591.406,A -85,B 0,C 180,E1 14057.089,E2 14057.089} C_VEL
LIN {X 0,Y 479.735,Z 588.146,A -85,B 0,C 180,E1 14053.745,E2 14053.745} C_VEL
LIN {X 0,Y 473.752,Z 586.463,A -85,B 0,C 180,E1 14049.966,E2 14049.966} C_VEL
LIN {X 0,Y 469.145,Z 588.495,A -85,B 0,C 180,E1 14045.995,E2 14045.995} C_VEL
LIN {X 0,Y 467.114,Z 591.489,A -85,B 0,C 180,E1 14043.313,E2 14043.313} C_VEL
LIN {X 0,Y 465.831,Z 596.462,A -85,B 0,C 180,E1 14040.246,E2 14040.246} C_VEL
LIN {X 0,Y 465.625,Z 603.576,A -85,B 0,C 180,E1 14037.169,E2 14037.169} C_VEL
LIN {X 0,Y 463.054,Z 636.252,A -85,B 0,C 180,E1 14034.703,E2 14034.703} C_VEL
LIN {X 0,Y 460.697,Z 671.163,A -85,B 0,C 180,E1 14032.227,E2 14032.227} C_VEL
LIN {X 0,Y 458.947,Z 700.452,A -85,B 0,C 180,E1 14030.105,E2 14030.105} C_VEL
LIN {X 0,Y 458.067,Z 726.682,A -85,B 0,C 180,E1 14027.925,E2 14027.925} C_VEL
LIN {X 0,Y 458.143,Z 751.981,A -85,B 0,C 180,E1 14025.529,E2 14025.529} C_VEL
LIN {X 0,Y 459.19,Z 772.76,A -85,B 0,C 180,E1 14023.313,E2 14023.313} C_VEL
LIN {X 0,Y 461.239,Z 792.123,A -85,B 0,C 180,E1 14021.04,E2 14021.04} C_VEL
LIN {X 0,Y 462.831,Z 802.878,A -85,B 0,C 180,E1 14019.709,E2 14019.709} C_VEL
LIN {X 0,Y 454.245,Z 843.477,A -85,B 0,C 180,E1 14018.787,E2 14018.787} C_VEL
LIN {X 0,Y 445.234,Z 880.201,A -85,B 0,C 180,E1 14017.785,E2 14017.785} C_VEL
LIN {X 0,Y 435.909,Z 915.267,A -85,B 0,C 180,E1 14016.56,E2 14016.56} C_VEL
LIN {X 0,Y 426.491,Z 948.186,A -85,B 0,C 180,E1 14015.13,E2 14015.13} C_VEL
LIN {X 0,Y 417.834,Z 976.311,A -85,B 0,C 180,E1 14013.656,E2 14013.656} C_VEL
LIN {X 0,Y 409.893,Z 998.76,A -85,B 0,C 180,E1 14012.23,E2 14012.23} C_VEL
LIN {X 0,Y 401.551,Z 1019.924,A -85,B 0,C 180,E1 14010.631,E2 14010.631} C_VEL
LIN {X 0,Y 392.042,Z 1041.295,A -85,B 0,C 180,E1 14008.689,E2 14008.689} C_VEL
LIN {X 0,Y 382.334,Z 1061.081,A -85,B 0,C 180,E1 14006.534,E2 14006.534} C_VEL
LIN {X 0,Y 372.56,Z 1079.624,A -85,B 0,C 180,E1 14004.142,E2 14004.142} C_VEL
LIN {X 0,Y 362.283,Z 1097.739,A -85,B 0,C 180,E1 14001.355,E2 14001.355} C_VEL
LIN {X 0,Y 352.752,Z 1113.454,A -85,B 0,C 180,E1 13998.441,E2 13998.441} C_VEL
LIN {X 0,Y 342.716,Z 1129.417,A -85,B 0,C 180,E1 13994.91,E2 13994.91} C_VEL
LIN {X 0,Y 333.823,Z 1143.181,A -85,B 0,C 180,E1 13991.217,E2 13991.217} C_VEL
LIN {X 0,Y 325.751,Z 1155.587,A -85,B 0,C 180,E1 13987.203,E2 13987.203} C_VEL
LIN {X 0,Y 318.529,Z 1166.904,A -85,B 0,C 180,E1 13982.675,E2 13982.675} C_VEL
LIN {X 0,Y 313.051,Z 1175.991,A -85,B 0,C 180,E1 13978.17,E2 13978.17} C_VEL
LIN {X 0,Y 308.802,Z 1183.937,A -85,B 0,C 180,E1 13973.265,E2 13973.265} C_VEL
LIN {X 0,Y 305.957,Z 1190.403,A -85,B 0,C 180,E1 13968.085,E2 13968.085} C_VEL
LIN {X 0,Y 304.572,Z 1194.857,A -85,B 0,C 180,E1 13963.283,E2 13963.283} C_VEL
LIN {X 0,Y 304.065,Z 1197.782,A -85,B 0,C 180,E1 13958.698,E2 13958.698} C_VEL
LIN {X 0,Y 303.973,Z 1199.402,A -85,B 0,C 180,E1 13954.337,E2 13954.337} C_VEL
LIN {X 0,Y 303.984,Z 1199.98,A -85,B 0,C 180,E1 13950.186,E2 13950.186} C_VEL
LIN {X 0,Y 303.976,Z 1199.491,A -85,B 0,C 180,E1 13946.037,E2 13946.037} C_VEL
LIN {X 0,Y 304.048,Z 1197.986,A -85,B 0,C 180,E1 13941.678,E2 13941.678} C_VEL
LIN {X 0,Y 304.505,Z 1195.126,A -85,B 0,C 180,E1 13937.096,E2 13937.096} C_VEL
LIN {X 0,Y 305.81,Z 1190.796,A -85,B 0,C 180,E1 13932.295,E2 13932.295} C_VEL
LIN {X 0,Y 308.544,Z 1184.469,A -85,B 0,C 180,E1 13927.113,E2 13927.113} C_VEL
LIN {X 0,Y 312.703,Z 1176.612,A -85,B 0,C 180,E1 13922.168,E2 13922.168} C_VEL
LIN {X 0,Y 318.276,Z 1167.295,A -85,B 0,C 180,E1 13917.504,E2 13917.504} C_VEL
LIN {X 0,Y 325.434,Z 1156.025,A -85,B 0,C 180,E1 13912.97,E2 13912.97} C_VEL
LIN {X 0,Y 333.829,Z 1143.147,A -85,B 0,C 180,E1 13908.778,E2 13908.778} C_VEL
LIN {X 0,Y 342.72,Z 1129.355,A -85,B 0,C 180,E1 13905.085,E2 13905.085} C_VEL
LIN {X 0,Y 352.785,Z 1113.386,A -85,B 0,C 180,E1 13901.546,E2 13901.546} C_VEL
LIN {X 0,Y 363.073,Z 1096.271,A -85,B 0,C 180,E1 13898.416,E2 13898.416} C_VEL
LIN {X 0,Y 373.414,Z 1078.017,A -85,B 0,C 180,E1 13895.639,E2 13895.639} C_VEL
LIN {X 0,Y 383.535,Z 1058.662,A -85,B 0,C 180,E1 13893.188,E2 13893.188} C_VEL
LIN {X 0,Y 393.288,Z 1038.391,A -85,B 0,C 180,E1 13891.041,E2 13891.041} C_VEL
LIN {X 0,Y 402.525,Z 1017.359,A -85,B 0,C 180,E1 13889.172,E2 13889.172} C_VEL
LIN {X 0,Y 411.418,Z 994.604,A -85,B 0,C 180,E1 13887.49,E2 13887.49} C_VEL
LIN {X 0,Y 419.194,Z 971.767,A -85,B 0,C 180,E1 13886.095,E2 13886.095} C_VEL
LIN {X 0,Y 429.339,Z 938.055,A -85,B 0,C 180,E1 13884.409,E2 13884.409} C_VEL
LIN {X 0,Y 438.708,Z 904.737,A -85,B 0,C 180,E1 13883.049,E2 13883.049} C_VEL
LIN {X 0,Y 447.684,Z 870.156,A -85,B 0,C 180,E1 13881.919,E2 13881.919} C_VEL
LIN {X 0,Y 457.223,Z 829.712,A -85,B 0,C 180,E1 13880.895,E2 13880.895} C_VEL
LIN {X 0,Y 465.834,Z 785.91,A -85,B 0,C 180,E1 13879.939,E2 13879.939} C_VEL
LIN {X 0,Y 460.724,Z 797.545,A -85,B 0,C 180,E1 13879.277,E2 13879.277} C_VEL
LIN {X 0,Y 452.891,Z 815.77,A -85,B 0,C 180,E1 13878.359,E2 13878.359} C_VEL
LIN {X 0,Y 447.592,Z 827.082,A -85,B 0,C 180,E1 13877.678,E2 13877.678} C_VEL
LIN {X 0,Y 439.648,Z 844.398,A -85,B 0,C 180,E1 13876.733,E2 13876.733} C_VEL
LIN {X 0,Y 435.115,Z 853.622,A -85,B 0,C 180,E1 13876.144,E2 13876.144} C_VEL
LIN {X 0,Y 427.328,Z 869.801,A -85,B 0,C 180,E1 13875.193,E2 13875.193} C_VEL
LIN {X 0,Y 423.214,Z 877.938,A -85,B 0,C 180,E1 13874.643,E2 13874.643} C_VEL
LIN {X 0,Y 415.802,Z 892.893,A -85,B 0,C 180,E1 13873.706,E2 13873.706} C_VEL
LIN {X 0,Y 412.798,Z 898.671,A -85,B 0,C 180,E1 13873.304,E2 13873.304} C_VEL
LIN {X 0,Y 404.525,Z 915.609,A -85,B 0,C 180,E1 13872.309,E2 13872.309} C_VEL
LIN {X 0,Y 398.06,Z 929.522,A -85,B 0,C 180,E1 13871.74,E2 13871.74} C_VEL
LIN {X 0,Y 394.762,Z 936.403,A -85,B 0,C 180,E1 13871.408,E2 13871.408} C_VEL
LIN {X 0,Y 388.234,Z 949.546,A -85,B 0,C 180,E1 13870.837,E2 13870.837} C_VEL
LIN {X 0,Y 384.329,Z 956.676,A -85,B 0,C 180,E1 13870.442,E2 13870.442} C_VEL
LIN {X 0,Y 377.848,Z 968.05,A -85,B 0,C 180,E1 13869.857,E2 13869.857} C_VEL
LIN {X 0,Y 374.079,Z 974.124,A -85,B 0,C 180,E1 13869.484,E2 13869.484} C_VEL
LIN {X 0,Y 367.574,Z 984.214,A -85,B 0,C 180,E1 13868.833,E2 13868.833} C_VEL
LIN {X 0,Y 359.09,Z 996.387,A -85,B 0,C 180,E1 13867.931,E2 13867.931} C_VEL
LIN {X 0,Y 351.322,Z 1006.709,A -85,B 0,C 180,E1 13867.03,E2 13867.03} C_VEL
LIN {X 0,Y 343.904,Z 1015.935,A -85,B 0,C 180,E1 13866.081,E2 13866.081} C_VEL
LIN {X 0,Y 337.16,Z 1023.912,A -85,B 0,C 180,E1 13865.104,E2 13865.104} C_VEL
LIN {X 0,Y 331.389,Z 1030.438,A -85,B 0,C 180,E1 13864.153,E2 13864.153} C_VEL
LIN {X 0,Y 329.171,Z 1032.861,A -85,B 0,C 180,E1 13863.739,E2 13863.739} C_VEL
LIN {X 0,Y 325.432,Z 1036.815,A -85,B 0,C 180,E1 13862.994,E2 13862.994} C_VEL
LIN {X 0,Y 321.186,Z 1041.303,A -85,B 0,C 180,E1 13862.091,E2 13862.091} C_VEL
LIN {X 0,Y 320.194,Z 1042.612,A -85,B 0,C 180,E1 13861.74,E2 13861.74} C_VEL
LIN {X 0,Y 318.985,Z 1054.955,A -85,B 0,C 180,E1 13860.515,E2 13860.515} C_VEL
LIN {X 0,Y 317.657,Z 1065.938,A -85,B 0,C 180,E1 13859.15,E2 13859.15} C_VEL
LIN {X 0,Y 315.865,Z 1077.602,A -85,B 0,C 180,E1 13857.278,E2 13857.278} C_VEL
LIN {X 0,Y 314.398,Z 1085.673,A -85,B 0,C 180,E1 13855.622,E2 13855.622} C_VEL
LIN {X 0,Y 313.051,Z 1092.245,A -85,B 0,C 180,E1 13853.95,E2 13853.95} C_VEL
LIN {X 0,Y 311.712,Z 1098.068,A -85,B 0,C 180,E1 13852.072,E2 13852.072} C_VEL
LIN {X 0,Y 310.249,Z 1103.682,A -85,B 0,C 180,E1 13849.602,E2 13849.602} C_VEL
LIN {X 0,Y 309.162,Z 1106.949,A -85,B 0,C 180,E1 13847.295,E2 13847.295} C_VEL
LIN {X 0,Y 308.468,Z 1108.52,A -85,B 0,C 180,E1 13845.355,E2 13845.355} C_VEL
LIN {X 0,Y 307.949,Z 1109.015,A -85,B 0,C 180,E1 13843.309,E2 13843.309} C_VEL
LIN {X 0,Y 307.621,Z 1108.331,A -85,B 0,C 180,E1 13841.229,E2 13841.229} C_VEL
LIN {X 0,Y 307.503,Z 1106.113,A -85,B 0,C 180,E1 13838.842,E2 13838.842} C_VEL
LIN {X 0,Y 307.656,Z 1101.776,A -85,B 0,C 180,E1 13836.234,E2 13836.234} C_VEL
LIN {X 0,Y 308.03,Z 1096.518,A -85,B 0,C 180,E1 13834.052,E2 13834.052} C_VEL
LIN {X 0,Y 308.534,Z 1090.718,A -85,B 0,C 180,E1 13832.181,E2 13832.181} C_VEL
LIN {X 0,Y 309.253,Z 1083.341,A -85,B 0,C 180,E1 13830.244,E2 13830.244} C_VEL
LIN {X 0,Y 310.719,Z 1083.891,A -85,B 0,C 180,E1 13829.44,E2 13829.44} C_VEL
LIN {X 0,Y 312.441,Z 1083.974,A -85,B 0,C 180,E1 13828.772,E2 13828.772} C_VEL
LIN {X 0,Y 320.822,Z 1084.317,A -85,B 0,C 180,E1 13825.875,E2 13825.875} C_VEL
LIN {X 0,Y 332.03,Z 1083.731,A -85,B 0,C 180,E1 13822.966,E2 13822.966} C_VEL
LIN {X 0,Y 345.659,Z 1082.067,A -85,B 0,C 180,E1 13820.261,E2 13820.261} C_VEL
LIN {X 0,Y 354.13,Z 1080.609,A -85,B 0,C 180,E1 13818.899,E2 13818.899} C_VEL
LIN {X 0,Y 344.052,Z 1097.874,A -85,B 0,C 180,E1 13815.402,E2 13815.402} C_VEL
LIN {X 0,Y 335.443,Z 1112.354,A -85,B 0,C 180,E1 13811.892,E2 13811.892} C_VEL
LIN {X 0,Y 326.963,Z 1126.88,A -85,B 0,C 180,E1 13807.709,E2 13807.709} C_VEL
LIN {X 0,Y 320.467,Z 1138.344,A -85,B 0,C 180,E1 13803.739,E2 13803.739} C_VEL
LIN {X 0,Y 314.464,Z 1149.725,A -85,B 0,C 180,E1 13799.025,E2 13799.025} C_VEL
LIN {X 0,Y 310.444,Z 1158.129,A -85,B 0,C 180,E1 13794.755,E2 13794.755} C_VEL
LIN {X 0,Y 307.294,Z 1165.872,A -85,B 0,C 180,E1 13789.98,E2 13789.98} C_VEL
LIN {X 0,Y 305.426,Z 1171.54,A -85,B 0,C 180,E1 13785.379,E2 13785.379} C_VEL
LIN {X 0,Y 304.562,Z 1175.174,A -85,B 0,C 180,E1 13781.555,E2 13781.555} C_VEL
LIN {X 0,Y 304.161,Z 1177.789,A -85,B 0,C 180,E1 13777.748,E2 13777.748} C_VEL
LIN {X 0,Y 304.009,Z 1179.607,A -85,B 0,C 180,E1 13773.396,E2 13773.396} C_VEL
LIN {X 0,Y 303.984,Z 1179.932,A -85,B 0,C 180,E1 13769.06,E2 13769.06} C_VEL
LIN {X 0,Y 304.026,Z 1179.166,A -85,B 0,C 180,E1 13765.286,E2 13765.286} C_VEL
LIN {X 0,Y 304.198,Z 1177.486,A -85,B 0,C 180,E1 13761.644,E2 13761.644} C_VEL
LIN {X 0,Y 304.61,Z 1174.897,A -85,B 0,C 180,E1 13758.014,E2 13758.014} C_VEL
LIN {X 0,Y 305.575,Z 1171.04,A -85,B 0,C 180,E1 13754.049,E2 13754.049} C_VEL
LIN {X 0,Y 307.77,Z 1164.576,A -85,B 0,C 180,E1 13749.064,E2 13749.064} C_VEL
LIN {X 0,Y 310.678,Z 1157.622,A -85,B 0,C 180,E1 13744.863,E2 13744.863} C_VEL
LIN {X 0,Y 315.091,Z 1148.594,A -85,B 0,C 180,E1 13740.331,E2 13740.331} C_VEL
LIN {X 0,Y 320.876,Z 1137.625,A -85,B 0,C 180,E1 13735.885,E2 13735.885} C_VEL
LIN {X 0,Y 327.829,Z 1125.534,A -85,B 0,C 180,E1 13731.749,E2 13731.749} C_VEL
LIN {X 0,Y 336.057,Z 1111.373,A -85,B 0,C 180,E1 13727.749,E2 13727.749} C_VEL
LIN {X 0,Y 345.211,Z 1096.061,A -85,B 0,C 180,E1 13724.088,E2 13724.088} C_VEL
LIN {X 0,Y 354.656,Z 1079.789,A -85,B 0,C 180,E1 13720.85,E2 13720.85} C_VEL
LIN {X 0,Y 364.953,Z 1061.784,A -85,B 0,C 180,E1 13717.8,E2 13717.8} C_VEL
LIN {X 0,Y 365.302,Z 1061.13,A -85,B 0,C 180,E1 13717.702,E2 13717.702} C_VEL
LIN {X 0,Y 367.412,Z 1056.177,A -85,B 0,C 180,E1 13716.824,E2 13716.824} C_VEL
LIN {X 0,Y 370.81,Z 1043.683,A -85,B 0,C 180,E1 13714.21,E2 13714.21} C_VEL
LIN {X 0,Y 372.803,Z 1039.126,A -85,B 0,C 180,E1 13713.53,E2 13713.53} C_VEL
LIN {X 0,Y 382.986,Z 1019.443,A -85,B 0,C 180,E1 13711.264,E2 13711.264} C_VEL
LIN {X 0,Y 393.052,Z 998.788,A -85,B 0,C 180,E1 13709.238,E2 13709.238} C_VEL
LIN {X 0,Y 402.389,Z 977.634,A -85,B 0,C 180,E1 13707.494,E2 13707.494} C_VEL
LIN {X 0,Y 411.719,Z 954.336,A -85,B 0,C 180,E1 13705.876,E2 13705.876} C_VEL
LIN {X 0,Y 418.854,Z 934.168,A -85,B 0,C 180,E1 13704.693,E2 13704.693} C_VEL
LIN {X 0,Y 426.361,Z 910.425,A -85,B 0,C 180,E1 13703.52,E2 13703.52} C_VEL
LIN {X 0,Y 432.417,Z 887.642,A -85,B 0,C 180,E1 13702.592,E2 13702.592} C_VEL
LIN {X 0,Y 438.684,Z 859.52,A -85,B 0,C 180,E1 13701.674,E2 13701.674} C_VEL
LIN {X 0,Y 447.698,Z 815.677,A -85,B 0,C 180,E1 13700.539,E2 13700.539} C_VEL
LIN {X 0,Y 461,Z 746.786,A -85,B 0,C 180,E1 13699.017,E2 13699.017} C_VEL
LIN {X 0,Y 472.166,Z 680.774,A -85,B 0,C 180,E1 13697.728,E2 13697.728} C_VEL
LIN {X 0,Y 481.097,Z 618.472,A -85,B 0,C 180,E1 13696.633,E2 13696.633} C_VEL
LIN {X 0,Y 483.55,Z 598.401,A -85,B 0,C 180,E1 13696.278,E2 13696.278} C_VEL
LIN {X 0,Y 476.973,Z 595.515,A -85,B 0,C 180,E1 13692.839,E2 13692.839} C_VEL
LIN {X 0,Y 472.501,Z 594.41,A -85,B 0,C 180,E1 13689.87,E2 13689.87} C_VEL
LIN {X 0,Y 468.233,Z 596.368,A -85,B 0,C 180,E1 13686.129,E2 13686.129} C_VEL
LIN {X 0,Y 466.168,Z 599.374,A -85,B 0,C 180,E1 13683.443,E2 13683.443} C_VEL
LIN {X 0,Y 464.875,Z 604.275,A -85,B 0,C 180,E1 13680.431,E2 13680.431} C_VEL
LIN {X 0,Y 464.541,Z 610.371,A -85,B 0,C 180,E1 13677.81,E2 13677.81} C_VEL
LIN {X 0,Y 461.929,Z 639.978,A -85,B 0,C 180,E1 13675.57,E2 13675.57} C_VEL
LIN {X 0,Y 459.085,Z 674.981,A -85,B 0,C 180,E1 13673.081,E2 13673.081} C_VEL
LIN {X 0,Y 456.985,Z 704.456,A -85,B 0,C 180,E1 13670.936,E2 13670.936} C_VEL
LIN {X 0,Y 455.729,Z 731.609,A -85,B 0,C 180,E1 13668.664,E2 13668.664} C_VEL
LIN {X 0,Y 455.452,Z 756.982,A -85,B 0,C 180,E1 13666.236,E2 13666.236} C_VEL
LIN {X 0,Y 456.209,Z 778.02,A -85,B 0,C 180,E1 13663.969,E2 13663.969} C_VEL
LIN {X 0,Y 457.957,Z 797.593,A -85,B 0,C 180,E1 13661.642,E2 13661.642} C_VEL
LIN {X 0,Y 459.11,Z 806.302,A -85,B 0,C 180,E1 13660.559,E2 13660.559} C_VEL
LIN {X 0,Y 449.417,Z 850.078,A -85,B 0,C 180,E1 13659.555,E2 13659.555} C_VEL
LIN {X 0,Y 440.472,Z 885.555,A -85,B 0,C 180,E1 13658.563,E2 13658.563} C_VEL
LIN {X 0,Y 430.993,Z 919.99,A -85,B 0,C 180,E1 13657.328,E2 13657.328} C_VEL
LIN {X 0,Y 421.263,Z 952.997,A -85,B 0,C 180,E1 13655.865,E2 13655.865} C_VEL
LIN {X 0,Y 413.165,Z 978.576,A -85,B 0,C 180,E1 13654.508,E2 13654.508} C_VEL
LIN {X 0,Y 404.879,Z 1001.023,A -85,B 0,C 180,E1 13653.06,E2 13653.06} C_VEL
LIN {X 0,Y 395.864,Z 1022.615,A -85,B 0,C 180,E1 13651.383,E2 13651.383} C_VEL
LIN {X 0,Y 386.747,Z 1042.521,A -85,B 0,C 180,E1 13649.553,E2 13649.553} C_VEL
LIN {X 0,Y 376.895,Z 1061.952,A -85,B 0,C 180,E1 13647.415,E2 13647.415} C_VEL
LIN {X 0,Y 366.493,Z 1080.849,A -85,B 0,C 180,E1 13644.928,E2 13644.928} C_VEL
LIN {X 0,Y 356.499,Z 1097.908,A -85,B 0,C 180,E1 13642.269,E2 13642.269} C_VEL
LIN {X 0,Y 346.185,Z 1114.438,A -85,B 0,C 180,E1 13639.173,E2 13639.173} C_VEL
LIN {X 0,Y 336.748,Z 1128.799,A -85,B 0,C 180,E1 13635.932,E2 13635.932} C_VEL
LIN {X 0,Y 327.489,Z 1142.655,A -85,B 0,C 180,E1 13632.195,E2 13632.195} C_VEL
LIN {X 0,Y 319.063,Z 1155.094,A -85,B 0,C 180,E1 13628.12,E2 13628.12} C_VEL
LIN {X 0,Y 311.481,Z 1166.478,A -85,B 0,C 180,E1 13623.511,E2 13623.511} C_VEL
LIN {X 0,Y 305.449,Z 1176.032,A -85,B 0,C 180,E1 13618.681,E2 13618.681} C_VEL
LIN {X 0,Y 301.038,Z 1183.847,A -85,B 0,C 180,E1 13613.694,E2 13613.694} C_VEL
LIN {X 0,Y 298.136,Z 1190.082,A -85,B 0,C 180,E1 13608.576,E2 13608.576} C_VEL
LIN {X 0,Y 296.637,Z 1194.559,A -85,B 0,C 180,E1 13603.645,E2 13603.645} C_VEL
LIN {X 0,Y 296.079,Z 1197.507,A -85,B 0,C 180,E1 13598.934,E2 13598.934} C_VEL
LIN {X 0,Y 295.976,Z 1199.135,A -85,B 0,C 180,E1 13594.454,E2 13594.454} C_VEL
LIN {X 0,Y 295.988,Z 1199.718,A -85,B 0,C 180,E1 13590.191,E2 13590.191} C_VEL
LIN {X 0,Y 295.978,Z 1199.225,A -85,B 0,C 180,E1 13585.93,E2 13585.93} C_VEL
LIN {X 0,Y 296.06,Z 1197.712,A -85,B 0,C 180,E1 13581.452,E2 13581.452} C_VEL
LIN {X 0,Y 296.562,Z 1194.831,A -85,B 0,C 180,E1 13576.744,E2 13576.744} C_VEL
LIN {X 0,Y 298.013,Z 1190.38,A -85,B 0,C 180,E1 13571.718,E2 13571.718} C_VEL
LIN {X 0,Y 300.902,Z 1184.119,A -85,B 0,C 180,E1 13566.497,E2 13566.497} C_VEL
LIN {X 0,Y 305.448,Z 1176.025,A -85,B 0,C 180,E1 13561.319,E2 13561.319} C_VEL
LIN {X 0,Y 311.486,Z 1166.44,A -85,B 0,C 180,E1 13556.485,E2 13556.485} C_VEL
LIN {X 0,Y 319.092,Z 1155.013,A -85,B 0,C 180,E1 13551.862,E2 13551.862} C_VEL
LIN {X 0,Y 327.885,Z 1142.032,A -85,B 0,C 180,E1 13547.626,E2 13547.626} C_VEL
LIN {X 0,Y 337.66,Z 1127.427,A -85,B 0,C 180,E1 13543.733,E2 13543.733} C_VEL
LIN {X 0,Y 348.185,Z 1111.18,A -85,B 0,C 180,E1 13540.191,E2 13540.191} C_VEL
LIN {X 0,Y 358.953,Z 1093.746,A -85,B 0,C 180,E1 13537.052,E2 13537.052} C_VEL
LIN {X 0,Y 369.405,Z 1075.712,A -85,B 0,C 180,E1 13534.353,E2 13534.353} C_VEL
LIN {X 0,Y 379.657,Z 1056.532,A -85,B 0,C 180,E1 13531.963,E2 13531.963} C_VEL
LIN {X 0,Y 389.654,Z 1036.228,A -85,B 0,C 180,E1 13529.847,E2 13529.847} C_VEL
LIN {X 0,Y 399.504,Z 1014.125,A -85,B 0,C 180,E1 13527.931,E2 13527.931} C_VEL
LIN {X 0,Y 408.484,Z 991.434,A -85,B 0,C 180,E1 13526.299,E2 13526.299} C_VEL
LIN {X 0,Y 416.658,Z 967.627,A -85,B 0,C 180,E1 13524.888,E2 13524.888} C_VEL
LIN {X 0,Y 426.717,Z 934.484,A -85,B 0,C 180,E1 13523.284,E2 13523.284} C_VEL
LIN {X 0,Y 436.179,Z 901.099,A -85,B 0,C 180,E1 13521.967,E2 13521.967} C_VEL
LIN {X 0,Y 445.801,Z 864.273,A -85,B 0,C 180,E1 13520.818,E2 13520.818} C_VEL
LIN {X 0,Y 455.416,Z 823.348,A -85,B 0,C 180,E1 13519.824,E2 13519.824} C_VEL
LIN {X 0,Y 457.585,Z 812.941,A -85,B 0,C 180,E1 13519.582,E2 13519.582} C_VEL
LIN {X 0,Y 448.929,Z 831.314,A -85,B 0,C 180,E1 13518.539,E2 13518.539} C_VEL
LIN {X 0,Y 440.692,Z 848.799,A -85,B 0,C 180,E1 13517.594,E2 13517.594} C_VEL
LIN {X 0,Y 436.279,Z 857.601,A -85,B 0,C 180,E1 13517.049,E2 13517.049} C_VEL
LIN {X 0,Y 428.392,Z 873.587,A -85,B 0,C 180,E1 13516.126,E2 13516.126} C_VEL
LIN {X 0,Y 424.147,Z 881.736,A -85,B 0,C 180,E1 13515.59,E2 13515.59} C_VEL
LIN {X 0,Y 416.539,Z 896.705,A -85,B 0,C 180,E1 13514.669,E2 13514.669} C_VEL
LIN {X 0,Y 413.472,Z 902.51,A -85,B 0,C 180,E1 13514.28,E2 13514.28} C_VEL
LIN {X 0,Y 404.851,Z 919.729,A -85,B 0,C 180,E1 13513.318,E2 13513.318} C_VEL
